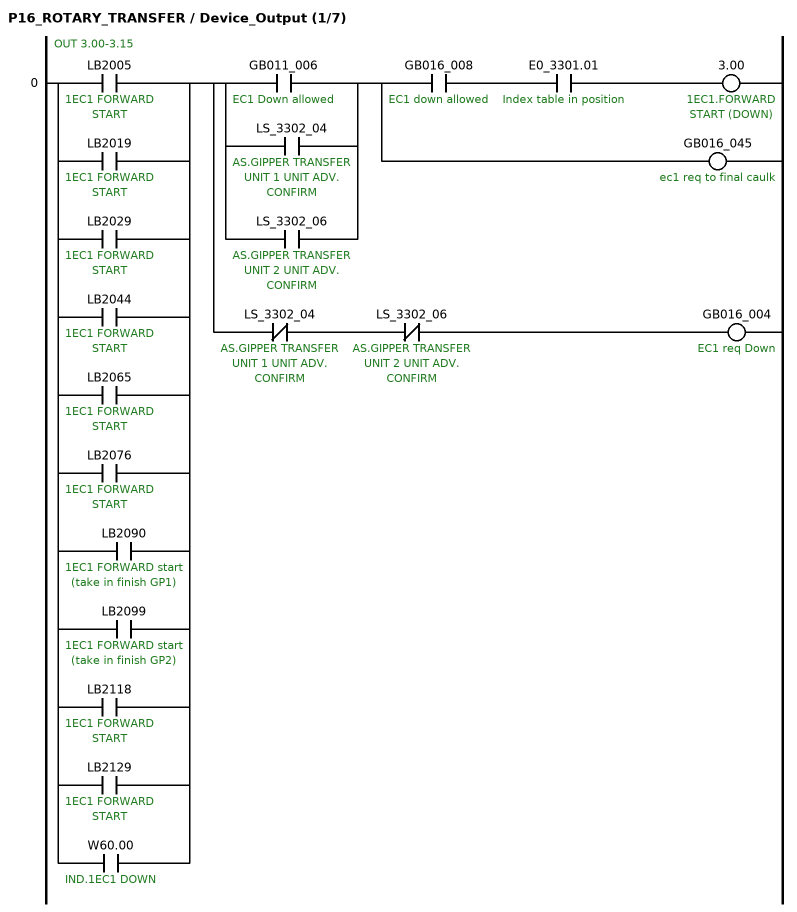
; [picture p264: P16_ROTARY_TRANSFER / Device_Output, rungs 0-0]
; rung 0: OUT 3.00-3.15
LD LB2005  ; 1EC1 FORWARD START
OR LB2019  ; 1EC1 FORWARD START
OR LB2029  ; 1EC1 FORWARD START
OR LB2044  ; 1EC1 FORWARD START
OR LB2065  ; 1EC1 FORWARD START
OR LB2076  ; 1EC1 FORWARD START
OR LB2090  ; 1EC1 FORWARD start (take in finish GP1)
OR LB2099  ; 1EC1 FORWARD start (take in finish GP2)
OR LB2118  ; 1EC1 FORWARD START
OR LB2129  ; 1EC1 FORWARD START
OR W60.00  ; IND.1EC1 DOWN
OUT TR0
LD GB011_006  ; EC1 Down allowed
OR LS_3302_04  ; AS.GIPPER TRANSFER UNIT 1 UNIT ADV. CONFIRM
OR LS_3302_06  ; AS.GIPPER TRANSFER UNIT 2 UNIT ADV. CONFIRM
ANDLD
OUT TR1
AND GB016_008  ; EC1 down allowed
AND E0_3301.01  ; Index table in position
OUT 3.00  ; 1EC1.FORWARD START (DOWN)
LD TR1
OUT GB016_045  ; ec1 req to final caulk
LD TR0
ANDNOT LS_3302_04  ; AS.GIPPER TRANSFER UNIT 1 UNIT ADV. CONFIRM
ANDNOT LS_3302_06  ; AS.GIPPER TRANSFER UNIT 2 UNIT ADV. CONFIRM
OUT GB016_004  ; EC1 req Down

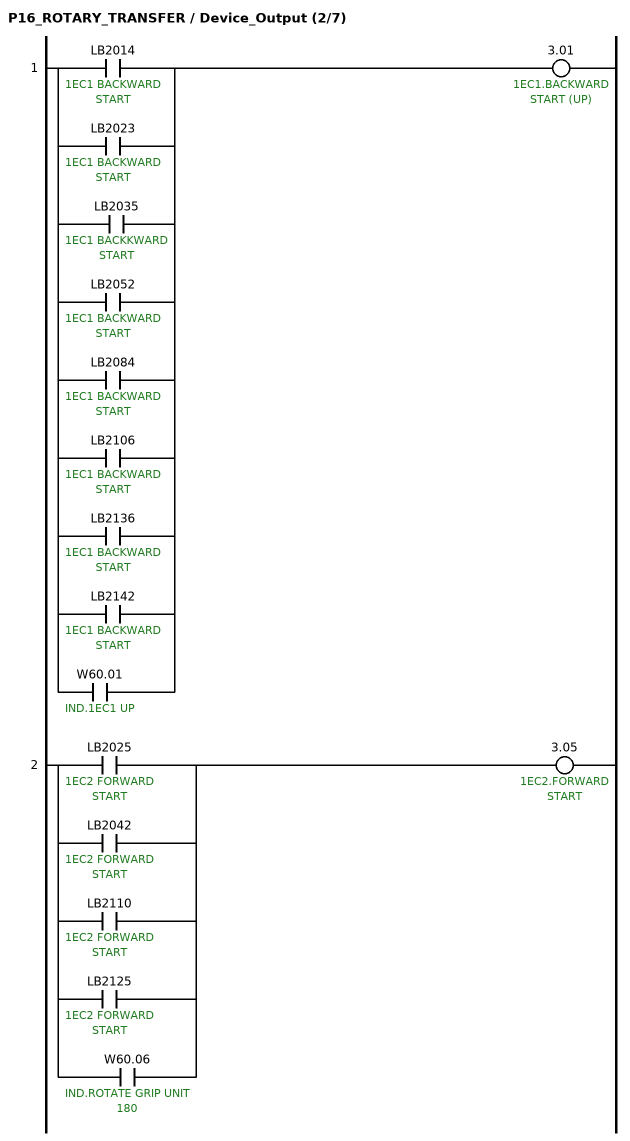
; rung 1
LD LB2014  ; 1EC1 BACKWARD START
OR LB2023  ; 1EC1 BACKWARD START
OR LB2035  ; 1EC1 BACKKWARD START
OR LB2052  ; 1EC1 BACKWARD START
OR LB2084  ; 1EC1 BACKWARD START
OR LB2106  ; 1EC1 BACKWARD START
OR LB2136  ; 1EC1 BACKWARD START
OR LB2142  ; 1EC1 BACKWARD START
OR W60.01  ; IND.1EC1 UP
OUT 3.01  ; 1EC1.BACKWARD START (UP)
; rung 2
LD LB2025  ; 1EC2 FORWARD START
OR LB2042  ; 1EC2 FORWARD START
OR LB2110  ; 1EC2 FORWARD START
OR LB2125  ; 1EC2 FORWARD START
OR W60.06  ; IND.ROTATE GRIP UNIT 180
OUT 3.05  ; 1EC2.FORWARD START

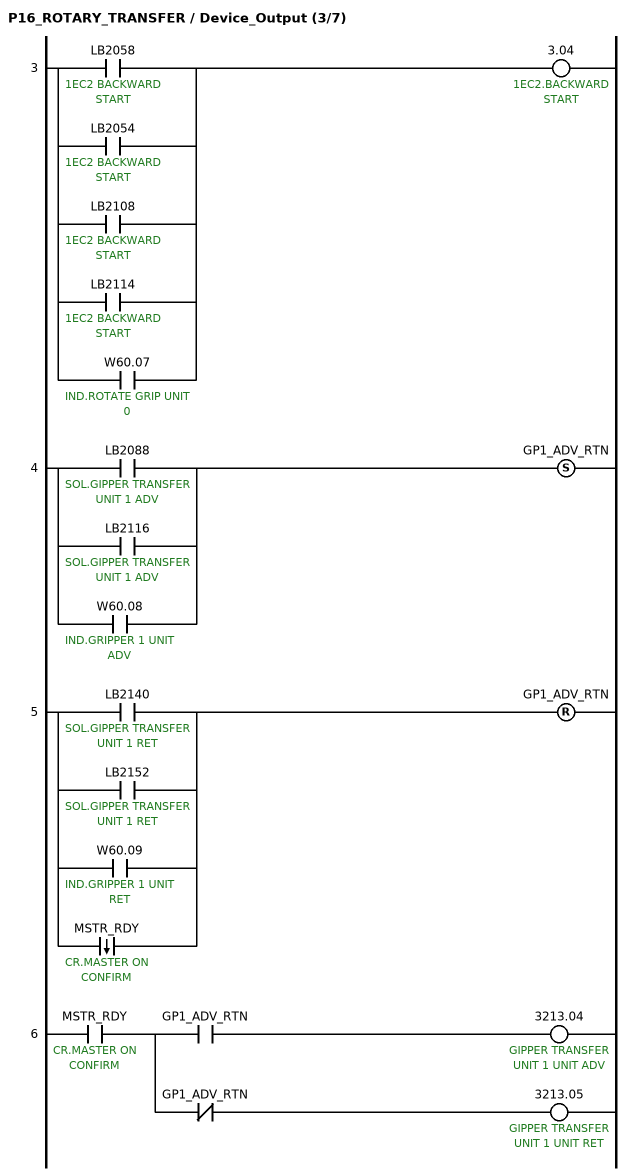
; rung 3
LD LB2058  ; 1EC2 BACKWARD START
OR LB2054  ; 1EC2 BACKWARD START
OR LB2108  ; 1EC2 BACKWARD START
OR LB2114  ; 1EC2 BACKWARD START
OR W60.07  ; IND.ROTATE GRIP UNIT 0
OUT 3.04  ; 1EC2.BACKWARD START
; rung 4
LD LB2088  ; SOL.GIPPER TRANSFER UNIT 1 ADV
OR LB2116  ; SOL.GIPPER TRANSFER UNIT 1 ADV
OR W60.08  ; IND.GRIPPER 1 UNIT ADV
SET GP1_ADV_RTN
; rung 5
LD LB2140  ; SOL.GIPPER TRANSFER UNIT 1 RET
OR LB2152  ; SOL.GIPPER TRANSFER UNIT 1 RET
OR W60.09  ; IND.GRIPPER 1 UNIT RET
%OR MSTR_RDY  ; CR.MASTER ON CONFIRM
RSET GP1_ADV_RTN
; rung 6
LD MSTR_RDY  ; CR.MASTER ON CONFIRM
OUT TR0
AND GP1_ADV_RTN
OUT 3213.04  ; GIPPER TRANSFER UNIT 1 UNIT ADV
LD TR0
ANDNOT GP1_ADV_RTN
OUT 3213.05  ; GIPPER TRANSFER UNIT 1 UNIT RET

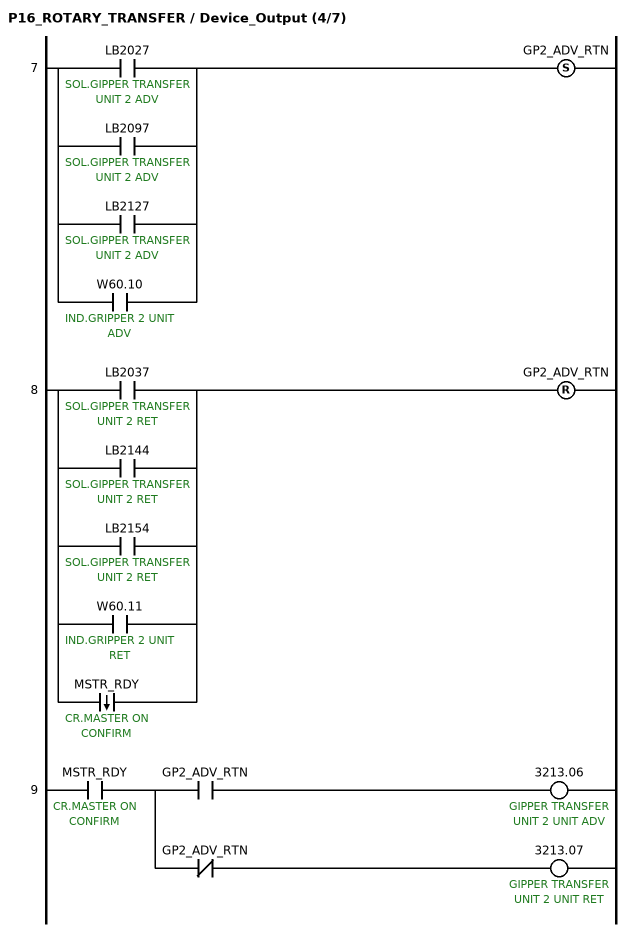
; rung 7
LD LB2027  ; SOL.GIPPER TRANSFER UNIT 2 ADV
OR LB2097  ; SOL.GIPPER TRANSFER UNIT 2 ADV
OR LB2127  ; SOL.GIPPER TRANSFER UNIT 2 ADV
OR W60.10  ; IND.GRIPPER 2 UNIT ADV
SET GP2_ADV_RTN
; rung 8
LD LB2037  ; SOL.GIPPER TRANSFER UNIT 2 RET
OR LB2144  ; SOL.GIPPER TRANSFER UNIT 2 RET
OR LB2154  ; SOL.GIPPER TRANSFER UNIT 2 RET
OR W60.11  ; IND.GRIPPER 2 UNIT RET
%OR MSTR_RDY  ; CR.MASTER ON CONFIRM
RSET GP2_ADV_RTN
; rung 9
LD MSTR_RDY  ; CR.MASTER ON CONFIRM
OUT TR0
AND GP2_ADV_RTN
OUT 3213.06  ; GIPPER TRANSFER UNIT 2 UNIT ADV
LD TR0
ANDNOT GP2_ADV_RTN
OUT 3213.07  ; GIPPER TRANSFER UNIT 2 UNIT RET

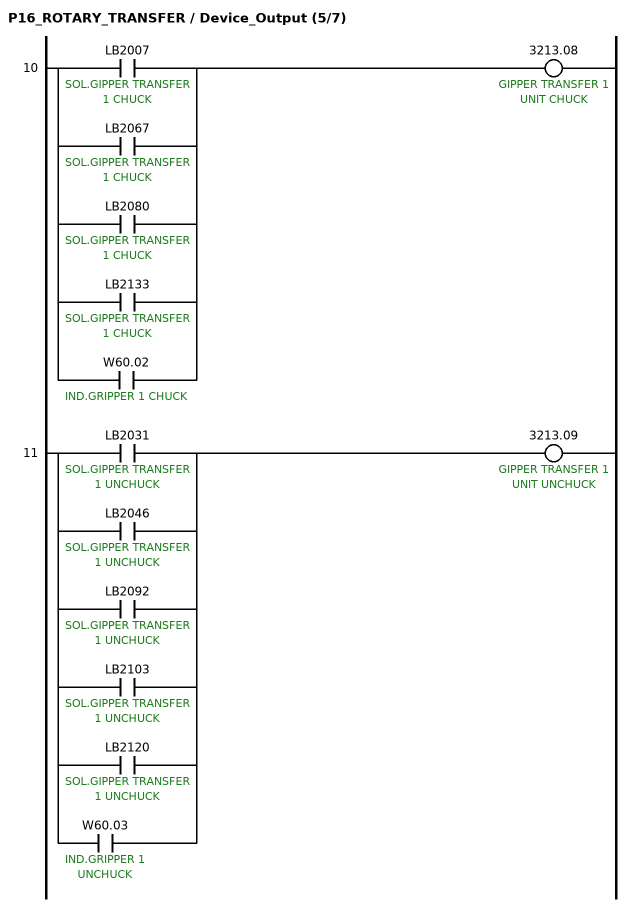
; rung 10
LD LB2007  ; SOL.GIPPER TRANSFER 1 CHUCK
OR LB2067  ; SOL.GIPPER TRANSFER 1 CHUCK
OR LB2080  ; SOL.GIPPER TRANSFER 1 CHUCK
OR LB2133  ; SOL.GIPPER TRANSFER 1 CHUCK
OR W60.02  ; IND.GRIPPER 1 CHUCK
OUT 3213.08  ; GIPPER TRANSFER 1 UNIT CHUCK
; rung 11
LD LB2031  ; SOL.GIPPER TRANSFER 1 UNCHUCK
OR LB2046  ; SOL.GIPPER TRANSFER 1 UNCHUCK
OR LB2092  ; SOL.GIPPER TRANSFER 1 UNCHUCK
OR LB2103  ; SOL.GIPPER TRANSFER 1 UNCHUCK
OR LB2120  ; SOL.GIPPER TRANSFER 1 UNCHUCK
OR W60.03  ; IND.GRIPPER 1 UNCHUCK
OUT 3213.09  ; GIPPER TRANSFER 1 UNIT UNCHUCK

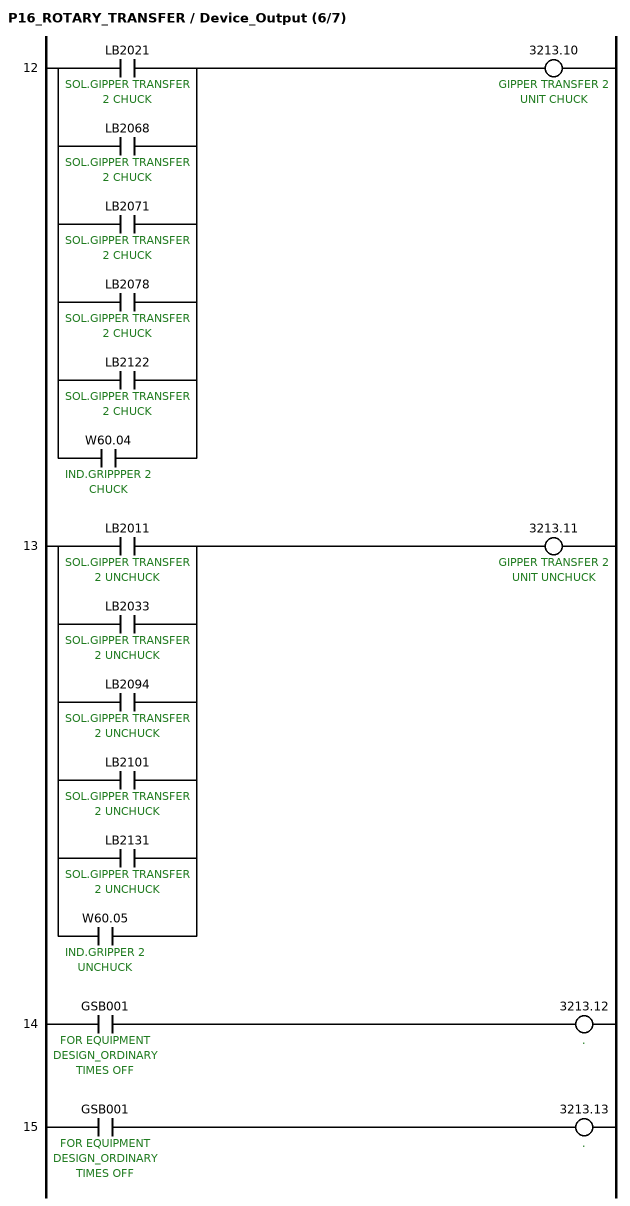
; rung 12
LD LB2021  ; SOL.GIPPER TRANSFER 2 CHUCK
OR LB2068  ; SOL.GIPPER TRANSFER 2 CHUCK
OR LB2071  ; SOL.GIPPER TRANSFER 2 CHUCK
OR LB2078  ; SOL.GIPPER TRANSFER 2 CHUCK
OR LB2122  ; SOL.GIPPER TRANSFER 2 CHUCK
OR W60.04  ; IND.GRIPPPER 2 CHUCK
OUT 3213.10  ; GIPPER TRANSFER 2 UNIT CHUCK
; rung 13
LD LB2011  ; SOL.GIPPER TRANSFER 2 UNCHUCK
OR LB2033  ; SOL.GIPPER TRANSFER 2 UNCHUCK
OR LB2094  ; SOL.GIPPER TRANSFER 2 UNCHUCK
OR LB2101  ; SOL.GIPPER TRANSFER 2 UNCHUCK
OR LB2131  ; SOL.GIPPER TRANSFER 2 UNCHUCK
OR W60.05  ; IND.GRIPPER 2 UNCHUCK
OUT 3213.11  ; GIPPER TRANSFER 2 UNIT UNCHUCK
; rung 14
LD GSB001  ; FOR EQUIPMENT DESIGN_ORDINARY TIMES OFF
OUT 3213.12  ; .
; rung 15
LD GSB001  ; FOR EQUIPMENT DESIGN_ORDINARY TIMES OFF
OUT 3213.13  ; .

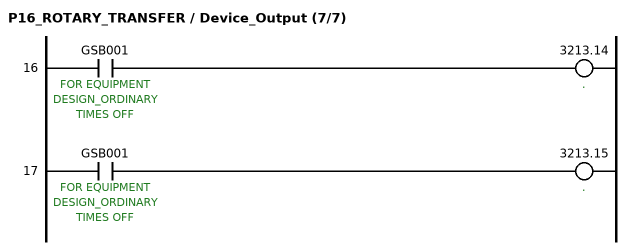
; rung 16
LD GSB001  ; FOR EQUIPMENT DESIGN_ORDINARY TIMES OFF
OUT 3213.14  ; .
; rung 17
LD GSB001  ; FOR EQUIPMENT DESIGN_ORDINARY TIMES OFF
OUT 3213.15  ; .

### Section Station_Output

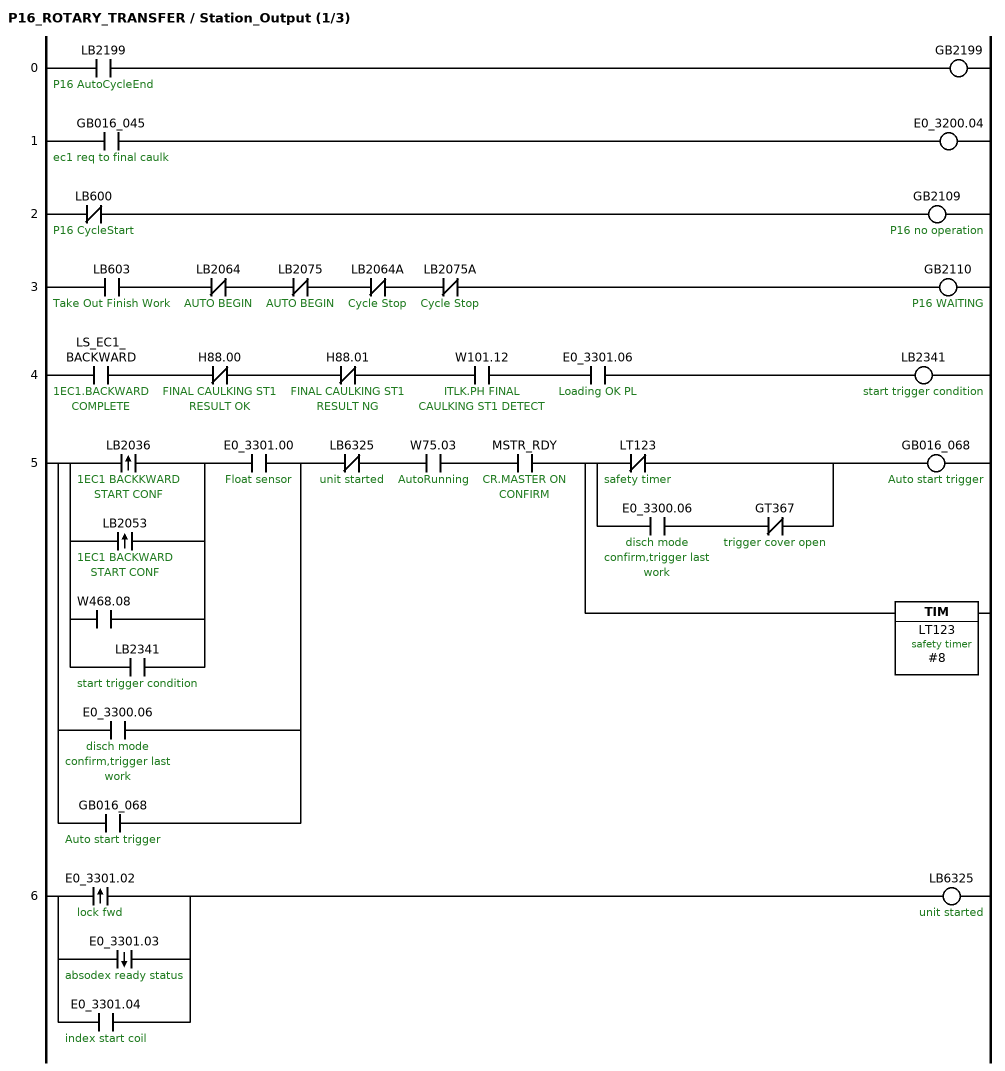
; rung 0
LD LB2199  ; P16 AutoCycleEnd
OUT GB2199
; rung 1
LD GB016_045  ; ec1 req to final caulk
OUT E0_3200.04
; rung 2
LDNOT LB600  ; P16 CycleStart
OUT GB2109  ; P16 no operation
; rung 3
LD LB603  ; Take Out Finish Work
ANDNOT LB2064  ; AUTO BEGIN
ANDNOT LB2075  ; AUTO BEGIN
ANDNOT LB2064A  ; Cycle Stop
ANDNOT LB2075A  ; Cycle Stop
OUT GB2110  ; P16 WAITING
; rung 4
LD LS_EC1_BACKWARD  ; 1EC1.BACKWARD COMPLETE
ANDNOT H88.00  ; FINAL CAULKING ST1 RESULT OK
ANDNOT H88.01  ; FINAL CAULKING ST1 RESULT NG
AND W101.12  ; ITLK.PH FINAL CAULKING ST1 DETECT
AND E0_3301.06  ; Loading OK PL
OUT LB2341  ; start trigger condition
; rung 5
@LD LB2036  ; 1EC1 BACKKWARD START CONF
@OR LB2053  ; 1EC1 BACKWARD START CONF
OR W468.08
OR LB2341  ; start trigger condition
AND E0_3301.00  ; Float sensor
OR E0_3300.06  ; disch mode confirm,trigger last work
OR GB016_068  ; Auto start trigger
ANDNOT LB6325  ; unit started
AND W75.03  ; AutoRunning
AND MSTR_RDY  ; CR.MASTER ON CONFIRM
OUT TR0
LDNOT LT123  ; safety timer
LD E0_3300.06  ; disch mode confirm,trigger last work
ANDNOT GT367  ; trigger cover open
ORLD
ANDLD
OUT GB016_068  ; Auto start trigger
LD TR0
TIM LT123 #8  ; safety timer
; rung 6
@LD E0_3301.02  ; lock fwd
%OR E0_3301.03  ; absodex ready status
OR E0_3301.04  ; index start coil
OUT LB6325  ; unit started

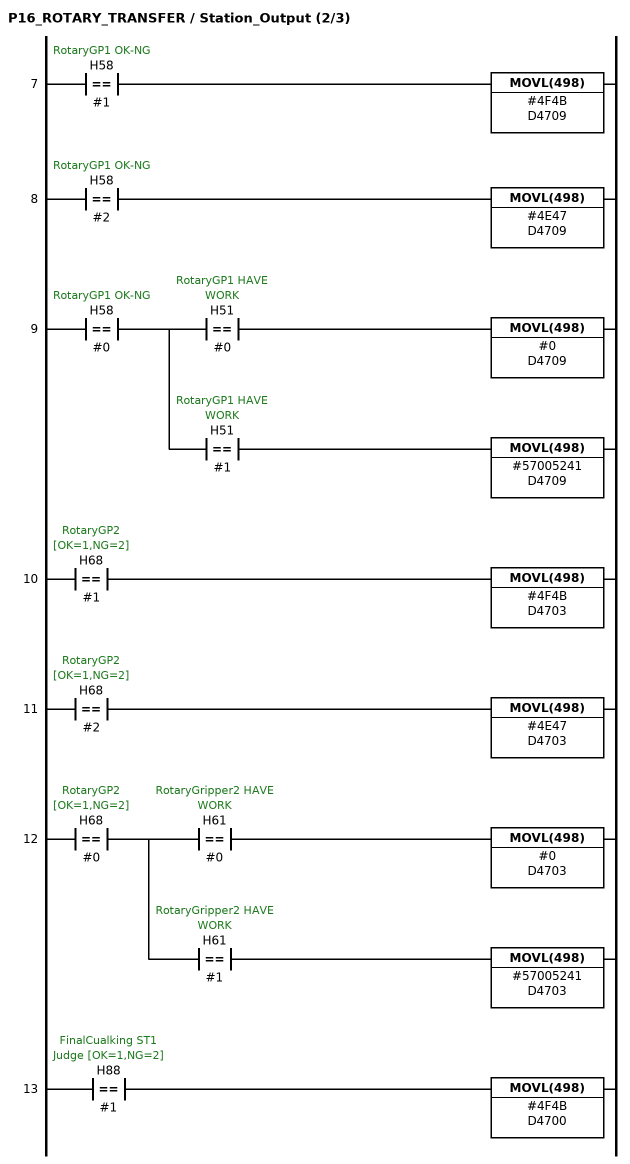
; rung 7
LD=(300) H58 #1  ; RotaryGP1 OK-NG
MOVL(498) #4F4B D4709
; rung 8
LD=(300) H58 #2  ; RotaryGP1 OK-NG
MOVL(498) #4E47 D4709
; rung 9
LD=(300) H58 #0  ; RotaryGP1 OK-NG
OUT TR0
AND=(300) H51 #0  ; RotaryGP1 HAVE WORK
MOVL(498) #0 D4709
LD TR0
AND=(300) H51 #1  ; RotaryGP1 HAVE WORK
MOVL(498) #57005241 D4709
; rung 10
LD=(300) H68 #1  ; RotaryGP2 [OK=1,NG=2]
MOVL(498) #4F4B D4703
; rung 11
LD=(300) H68 #2  ; RotaryGP2 [OK=1,NG=2]
MOVL(498) #4E47 D4703
; rung 12
LD=(300) H68 #0  ; RotaryGP2 [OK=1,NG=2]
OUT TR0
AND=(300) H61 #0  ; RotaryGripper2 HAVE WORK
MOVL(498) #0 D4703
LD TR0
AND=(300) H61 #1  ; RotaryGripper2 HAVE WORK
MOVL(498) #57005241 D4703
; rung 13
LD=(300) H88 #1  ; FinalCualking ST1 Judge [OK=1,NG=2]
MOVL(498) #4F4B D4700

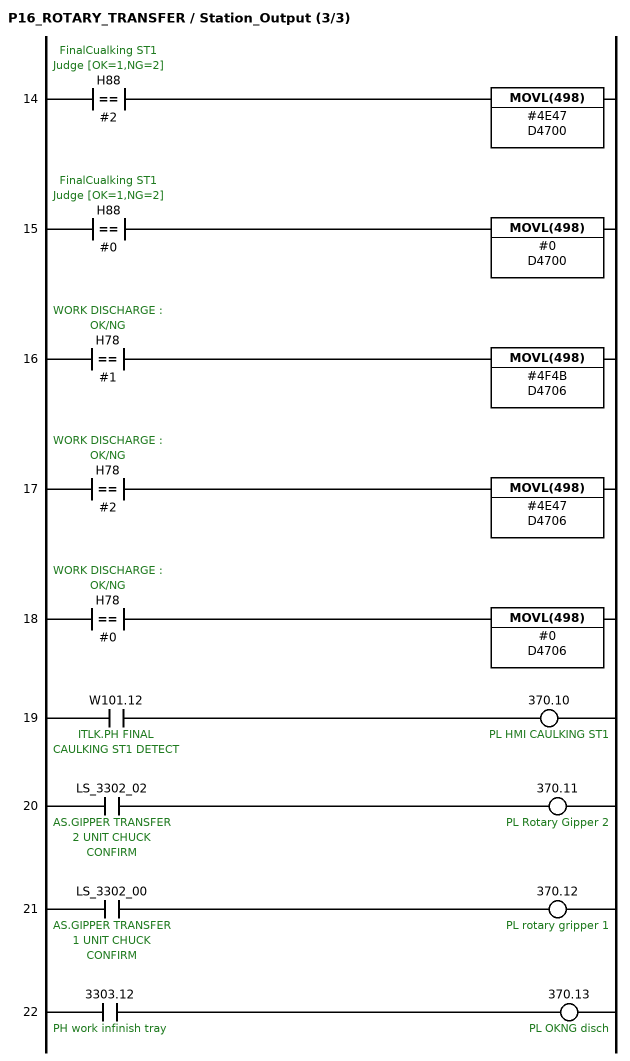
; rung 14
LD=(300) H88 #2  ; FinalCualking ST1 Judge [OK=1,NG=2]
MOVL(498) #4E47 D4700
; rung 15
LD=(300) H88 #0  ; FinalCualking ST1 Judge [OK=1,NG=2]
MOVL(498) #0 D4700
; rung 16
LD=(300) H78 #1  ; WORK DISCHARGE : OK/NG
MOVL(498) #4F4B D4706
; rung 17
LD=(300) H78 #2  ; WORK DISCHARGE : OK/NG
MOVL(498) #4E47 D4706
; rung 18
LD=(300) H78 #0  ; WORK DISCHARGE : OK/NG
MOVL(498) #0 D4706
; rung 19
LD W101.12  ; ITLK.PH FINAL CAULKING ST1 DETECT
OUT 370.10  ; PL HMI CAULKING ST1
; rung 20
LD LS_3302_02  ; AS.GIPPER TRANSFER 2 UNIT CHUCK CONFIRM
OUT 370.11  ; PL Rotary Gipper 2
; rung 21
LD LS_3302_00  ; AS.GIPPER TRANSFER 1 UNIT CHUCK CONFIRM
OUT 370.12  ; PL rotary gripper 1
; rung 22
LD 3303.12  ; PH work infinish tray
OUT 370.13  ; PL OKNG disch

### Section Individual

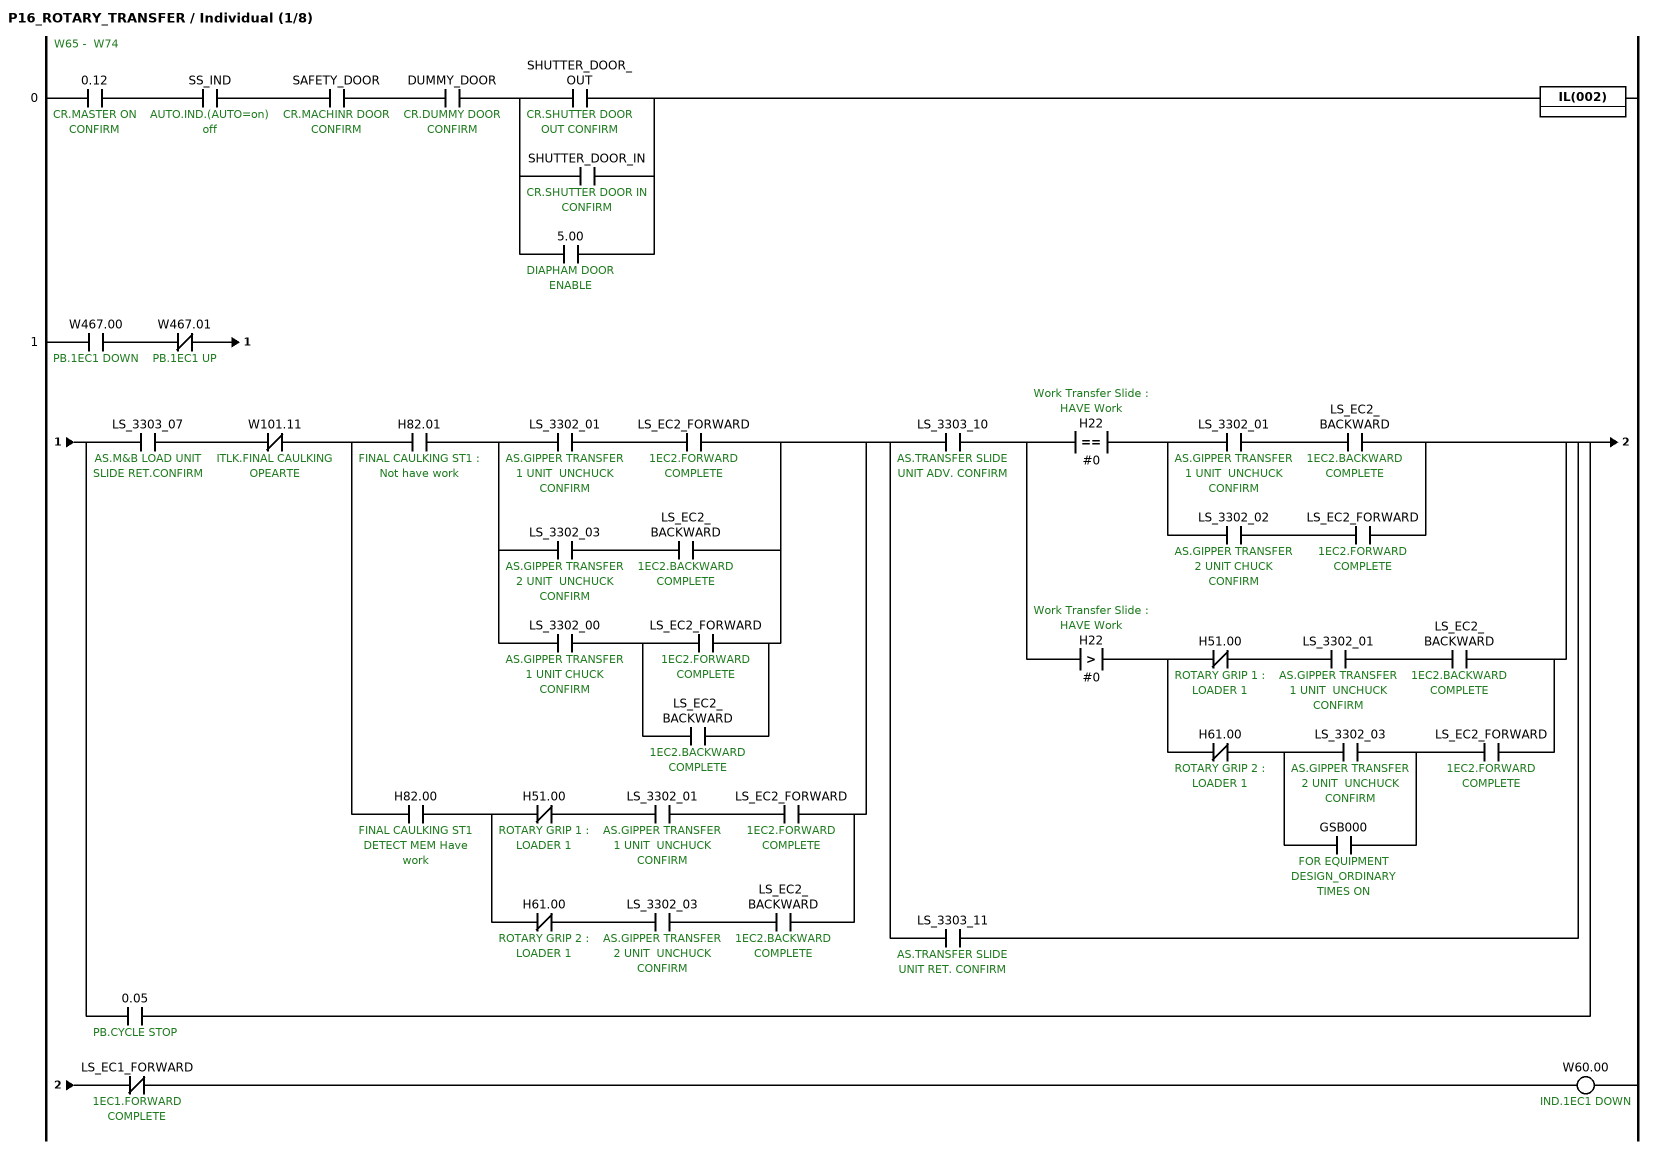
; rung 0: W65 -  W74
LD 0.12  ; CR.MASTER ON CONFIRM
AND SS_IND  ; AUTO.IND.(AUTO=on) off
AND SAFETY_DOOR  ; CR.MACHINR DOOR CONFIRM
AND DUMMY_DOOR  ; CR.DUMMY DOOR CONFIRM
LD SHUTTER_DOOR_OUT  ; CR.SHUTTER DOOR OUT CONFIRM
OR SHUTTER_DOOR_IN  ; CR.SHUTTER DOOR IN CONFIRM
OR 5.00  ; DIAPHAM DOOR ENABLE
ANDLD
IL(002)
; rung 1
LD W467.00  ; PB.1EC1 DOWN
ANDNOT W467.01  ; PB.1EC1 UP
LD LS_3303_07  ; AS.M&B LOAD UNIT SLIDE RET.CONFIRM
ANDNOT W101.11  ; ITLK.FINAL CAULKING OPEARTE
LD H82.01  ; FINAL CAULKING ST1 : Not have work
LD LS_3302_01  ; AS.GIPPER TRANSFER 1 UNIT  UNCHUCK CONFIRM
AND LS_EC2_FORWARD  ; 1EC2.FORWARD COMPLETE
LD LS_3302_03  ; AS.GIPPER TRANSFER 2 UNIT  UNCHUCK CONFIRM
AND LS_EC2_BACKWARD  ; 1EC2.BACKWARD COMPLETE
ORLD
LD LS_3302_00  ; AS.GIPPER TRANSFER 1 UNIT CHUCK CONFIRM
LD LS_EC2_FORWARD  ; 1EC2.FORWARD COMPLETE
OR LS_EC2_BACKWARD  ; 1EC2.BACKWARD COMPLETE
ANDLD
ORLD
ANDLD
LD H82.00  ; FINAL CAULKING ST1 DETECT MEM Have work
LDNOT H51.00  ; ROTARY GRIP 1 : LOADER 1
AND LS_3302_01  ; AS.GIPPER TRANSFER 1 UNIT  UNCHUCK CONFIRM
AND LS_EC2_FORWARD  ; 1EC2.FORWARD COMPLETE
LDNOT H61.00  ; ROTARY GRIP 2 : LOADER 1
AND LS_3302_03  ; AS.GIPPER TRANSFER 2 UNIT  UNCHUCK CONFIRM
AND LS_EC2_BACKWARD  ; 1EC2.BACKWARD COMPLETE
ORLD
ANDLD
ORLD
ANDLD
LD LS_3303_10  ; AS.TRANSFER SLIDE UNIT ADV. CONFIRM
LD=(300) H22 #0  ; Work Transfer Slide : HAVE Work
LD LS_3302_01  ; AS.GIPPER TRANSFER 1 UNIT  UNCHUCK CONFIRM
AND LS_EC2_BACKWARD  ; 1EC2.BACKWARD COMPLETE
LD LS_3302_02  ; AS.GIPPER TRANSFER 2 UNIT CHUCK CONFIRM
AND LS_EC2_FORWARD  ; 1EC2.FORWARD COMPLETE
ORLD
ANDLD
LD>(320) H22 #0  ; Work Transfer Slide : HAVE Work
LDNOT H51.00  ; ROTARY GRIP 1 : LOADER 1
AND LS_3302_01  ; AS.GIPPER TRANSFER 1 UNIT  UNCHUCK CONFIRM
AND LS_EC2_BACKWARD  ; 1EC2.BACKWARD COMPLETE
LDNOT H61.00  ; ROTARY GRIP 2 : LOADER 1
LD LS_3302_03  ; AS.GIPPER TRANSFER 2 UNIT  UNCHUCK CONFIRM
OR GSB000  ; FOR EQUIPMENT DESIGN_ORDINARY TIMES ON
ANDLD
AND LS_EC2_FORWARD  ; 1EC2.FORWARD COMPLETE
ORLD
ANDLD
ORLD
ANDLD
OR LS_3303_11  ; AS.TRANSFER SLIDE UNIT RET. CONFIRM
ANDLD
OR 0.05  ; PB.CYCLE STOP
ANDLD
ANDNOT LS_EC1_FORWARD  ; 1EC1.FORWARD COMPLETE
OUT W60.00  ; IND.1EC1 DOWN

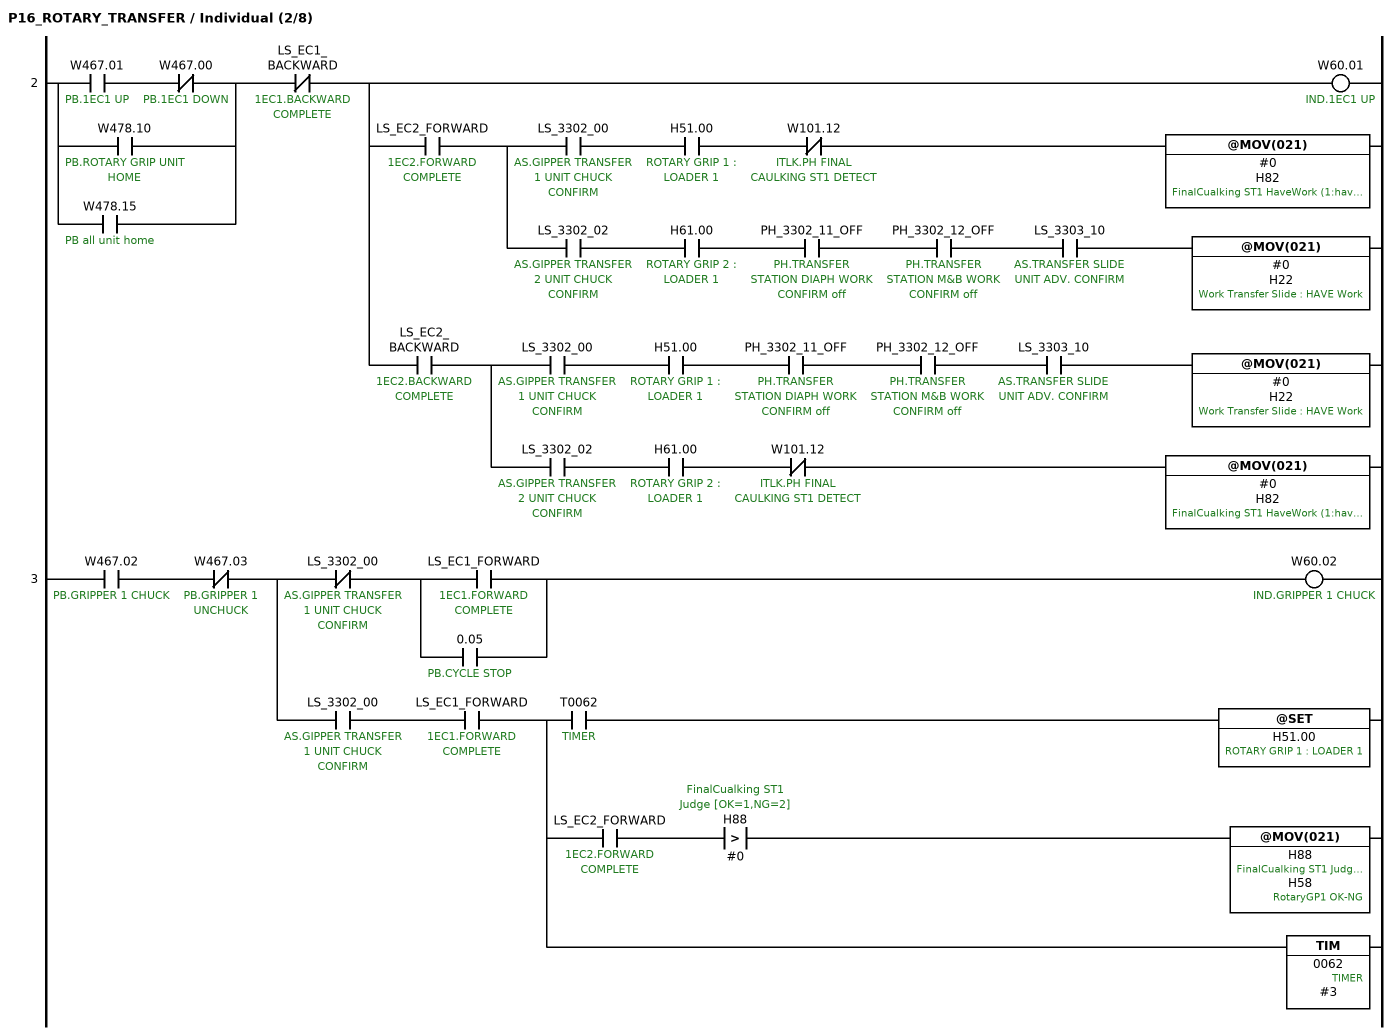
; rung 2
LD W467.01  ; PB.1EC1 UP
ANDNOT W467.00  ; PB.1EC1 DOWN
LD W478.10  ; PB.ROTARY GRIP UNIT HOME
OR W478.15  ; PB all unit home
ORLD
ANDNOT LS_EC1_BACKWARD  ; 1EC1.BACKWARD COMPLETE
OUT TR0
OUT W60.01  ; IND.1EC1 UP
AND LS_EC2_FORWARD  ; 1EC2.FORWARD COMPLETE
OUT TR1
AND LS_3302_00  ; AS.GIPPER TRANSFER 1 UNIT CHUCK CONFIRM
AND H51.00  ; ROTARY GRIP 1 : LOADER 1
ANDNOT W101.12  ; ITLK.PH FINAL CAULKING ST1 DETECT
@MOV(021) #0 H82  ; FinalCualking ST1 HaveWork (1:have work 2:no work)
LD TR1
AND LS_3302_02  ; AS.GIPPER TRANSFER 2 UNIT CHUCK CONFIRM
AND H61.00  ; ROTARY GRIP 2 : LOADER 1
AND PH_3302_11_OFF  ; PH.TRANSFER STATION DIAPH WORK CONFIRM off
AND PH_3302_12_OFF  ; PH.TRANSFER STATION M&B WORK CONFIRM off
AND LS_3303_10  ; AS.TRANSFER SLIDE UNIT ADV. CONFIRM
@MOV(021) #0 H22  ; Work Transfer Slide : HAVE Work
LD TR0
AND LS_EC2_BACKWARD  ; 1EC2.BACKWARD COMPLETE
OUT TR0
AND LS_3302_00  ; AS.GIPPER TRANSFER 1 UNIT CHUCK CONFIRM
AND H51.00  ; ROTARY GRIP 1 : LOADER 1
AND PH_3302_11_OFF  ; PH.TRANSFER STATION DIAPH WORK CONFIRM off
AND PH_3302_12_OFF  ; PH.TRANSFER STATION M&B WORK CONFIRM off
AND LS_3303_10  ; AS.TRANSFER SLIDE UNIT ADV. CONFIRM
@MOV(021) #0 H22  ; Work Transfer Slide : HAVE Work
LD TR0
AND LS_3302_02  ; AS.GIPPER TRANSFER 2 UNIT CHUCK CONFIRM
AND H61.00  ; ROTARY GRIP 2 : LOADER 1
ANDNOT W101.12  ; ITLK.PH FINAL CAULKING ST1 DETECT
@MOV(021) #0 H82  ; FinalCualking ST1 HaveWork (1:have work 2:no work)
; rung 3
LD W467.02  ; PB.GRIPPER 1 CHUCK
ANDNOT W467.03  ; PB.GRIPPER 1 UNCHUCK
OUT TR0
ANDNOT LS_3302_00  ; AS.GIPPER TRANSFER 1 UNIT CHUCK CONFIRM
LD LS_EC1_FORWARD  ; 1EC1.FORWARD COMPLETE
OR 0.05  ; PB.CYCLE STOP
ANDLD
OUT W60.02  ; IND.GRIPPER 1 CHUCK
LD TR0
AND LS_3302_00  ; AS.GIPPER TRANSFER 1 UNIT CHUCK CONFIRM
AND LS_EC1_FORWARD  ; 1EC1.FORWARD COMPLETE
OUT TR0
AND T0062  ; TIMER
@SET H51.00  ; ROTARY GRIP 1 : LOADER 1
LD TR0
AND LS_EC2_FORWARD  ; 1EC2.FORWARD COMPLETE
AND>(320) H88 #0  ; FinalCualking ST1 Judge [OK=1,NG=2]
@MOV(021) H88 H58  ; FinalCualking ST1 Judge [OK=1,NG=2], RotaryGP1 OK-NG
LD TR0
TIM 0062 #3  ; TIMER

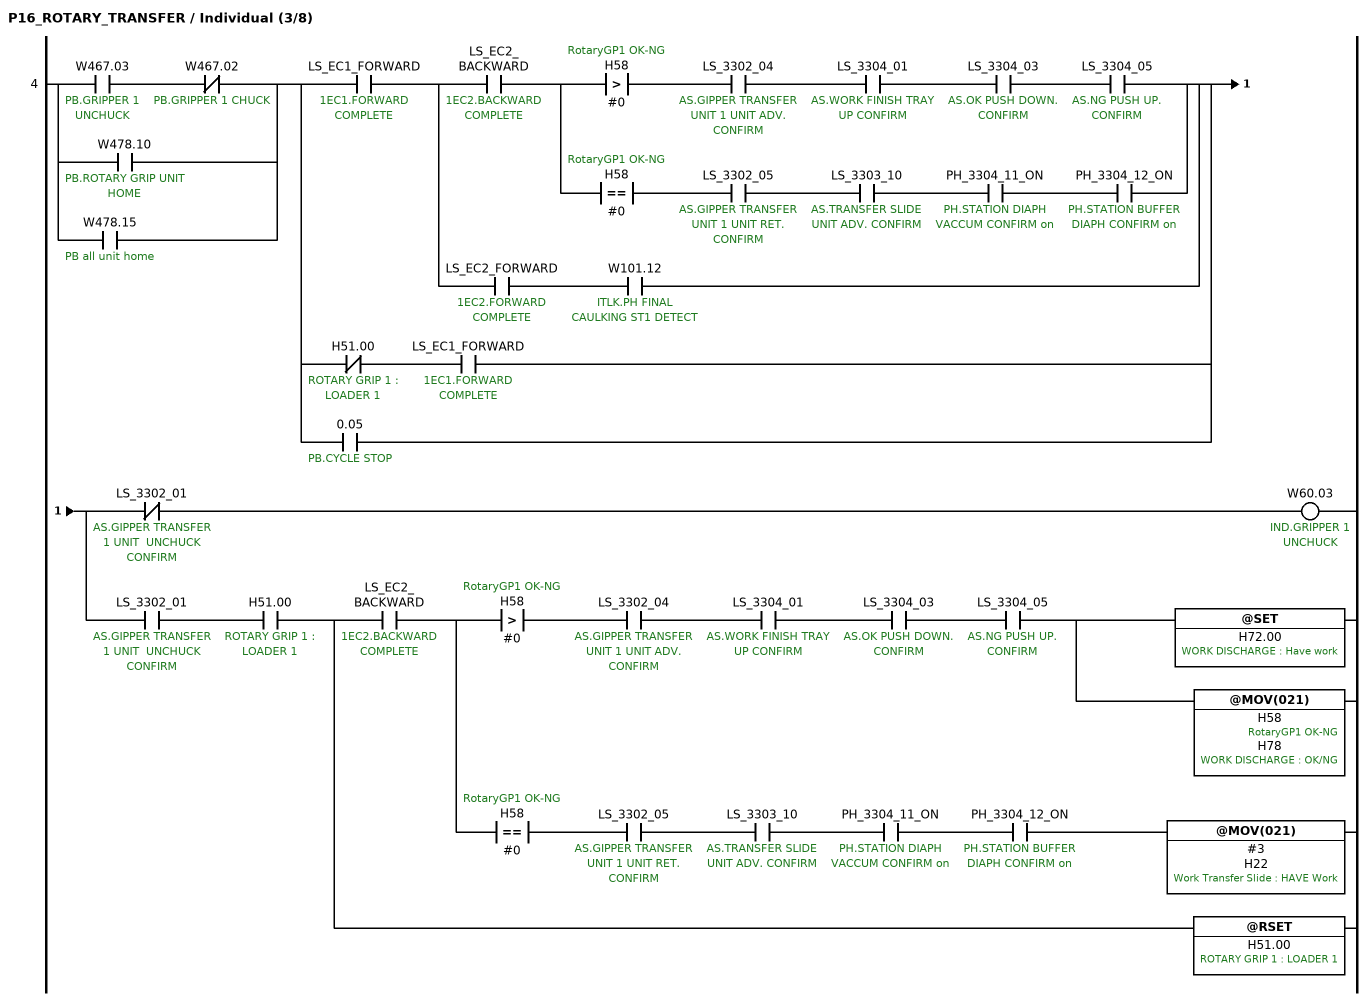
; rung 4
LD W467.03  ; PB.GRIPPER 1 UNCHUCK
ANDNOT W467.02  ; PB.GRIPPER 1 CHUCK
OR W478.10  ; PB.ROTARY GRIP UNIT HOME
OR W478.15  ; PB all unit home
LD LS_EC1_FORWARD  ; 1EC1.FORWARD COMPLETE
LD LS_EC2_BACKWARD  ; 1EC2.BACKWARD COMPLETE
LD>(320) H58 #0  ; RotaryGP1 OK-NG
AND LS_3302_04  ; AS.GIPPER TRANSFER UNIT 1 UNIT ADV. CONFIRM
AND LS_3304_01  ; AS.WORK FINISH TRAY UP CONFIRM
AND LS_3304_03  ; AS.OK PUSH DOWN. CONFIRM
AND LS_3304_05  ; AS.NG PUSH UP. CONFIRM
LD=(300) H58 #0  ; RotaryGP1 OK-NG
AND LS_3302_05  ; AS.GIPPER TRANSFER UNIT 1 UNIT RET. CONFIRM
AND LS_3303_10  ; AS.TRANSFER SLIDE UNIT ADV. CONFIRM
AND PH_3304_11_ON  ; PH.STATION DIAPH VACCUM CONFIRM on
AND PH_3304_12_ON  ; PH.STATION BUFFER DIAPH CONFIRM on
ORLD
ANDLD
LD LS_EC2_FORWARD  ; 1EC2.FORWARD COMPLETE
AND W101.12  ; ITLK.PH FINAL CAULKING ST1 DETECT
ORLD
ANDLD
LDNOT H51.00  ; ROTARY GRIP 1 : LOADER 1
AND LS_EC1_FORWARD  ; 1EC1.FORWARD COMPLETE
ORLD
OR 0.05  ; PB.CYCLE STOP
ANDLD
OUT TR0
ANDNOT LS_3302_01  ; AS.GIPPER TRANSFER 1 UNIT  UNCHUCK CONFIRM
OUT W60.03  ; IND.GRIPPER 1 UNCHUCK
LD TR0
AND LS_3302_01  ; AS.GIPPER TRANSFER 1 UNIT  UNCHUCK CONFIRM
AND H51.00  ; ROTARY GRIP 1 : LOADER 1
OUT TR0
AND LS_EC2_BACKWARD  ; 1EC2.BACKWARD COMPLETE
OUT TR1
AND>(320) H58 #0  ; RotaryGP1 OK-NG
AND LS_3302_04  ; AS.GIPPER TRANSFER UNIT 1 UNIT ADV. CONFIRM
AND LS_3304_01  ; AS.WORK FINISH TRAY UP CONFIRM
AND LS_3304_03  ; AS.OK PUSH DOWN. CONFIRM
AND LS_3304_05  ; AS.NG PUSH UP. CONFIRM
@SET H72.00  ; WORK DISCHARGE : Have work
@MOV(021) H58 H78  ; RotaryGP1 OK-NG, WORK DISCHARGE : OK/NG
LD TR1
AND=(300) H58 #0  ; RotaryGP1 OK-NG
AND LS_3302_05  ; AS.GIPPER TRANSFER UNIT 1 UNIT RET. CONFIRM
AND LS_3303_10  ; AS.TRANSFER SLIDE UNIT ADV. CONFIRM
AND PH_3304_11_ON  ; PH.STATION DIAPH VACCUM CONFIRM on
AND PH_3304_12_ON  ; PH.STATION BUFFER DIAPH CONFIRM on
@MOV(021) #3 H22  ; Work Transfer Slide : HAVE Work
LD TR0
@RSET H51.00  ; ROTARY GRIP 1 : LOADER 1

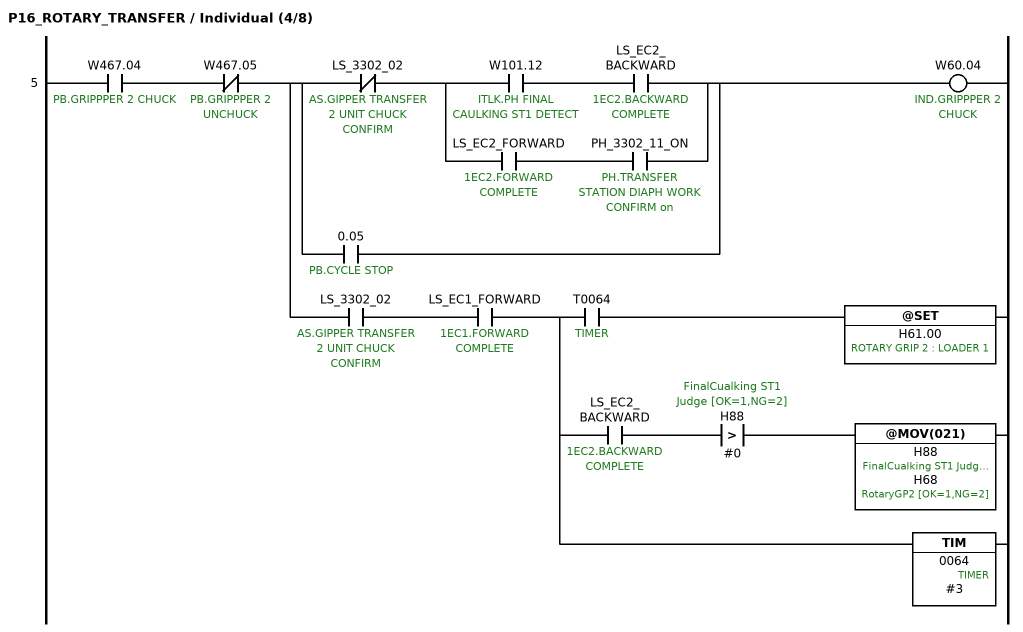
; rung 5
LD W467.04  ; PB.GRIPPPER 2 CHUCK
ANDNOT W467.05  ; PB.GRIPPPER 2 UNCHUCK
OUT TR0
LDNOT LS_3302_02  ; AS.GIPPER TRANSFER 2 UNIT CHUCK CONFIRM
LD W101.12  ; ITLK.PH FINAL CAULKING ST1 DETECT
AND LS_EC2_BACKWARD  ; 1EC2.BACKWARD COMPLETE
LD LS_EC2_FORWARD  ; 1EC2.FORWARD COMPLETE
AND PH_3302_11_ON  ; PH.TRANSFER STATION DIAPH WORK CONFIRM on
ORLD
ANDLD
OR 0.05  ; PB.CYCLE STOP
ANDLD
OUT W60.04  ; IND.GRIPPPER 2 CHUCK
LD TR0
AND LS_3302_02  ; AS.GIPPER TRANSFER 2 UNIT CHUCK CONFIRM
AND LS_EC1_FORWARD  ; 1EC1.FORWARD COMPLETE
OUT TR0
AND T0064  ; TIMER
@SET H61.00  ; ROTARY GRIP 2 : LOADER 1
LD TR0
AND LS_EC2_BACKWARD  ; 1EC2.BACKWARD COMPLETE
AND>(320) H88 #0  ; FinalCualking ST1 Judge [OK=1,NG=2]
@MOV(021) H88 H68  ; FinalCualking ST1 Judge [OK=1,NG=2], RotaryGP2 [OK=1,NG=2]
LD TR0
TIM 0064 #3  ; TIMER

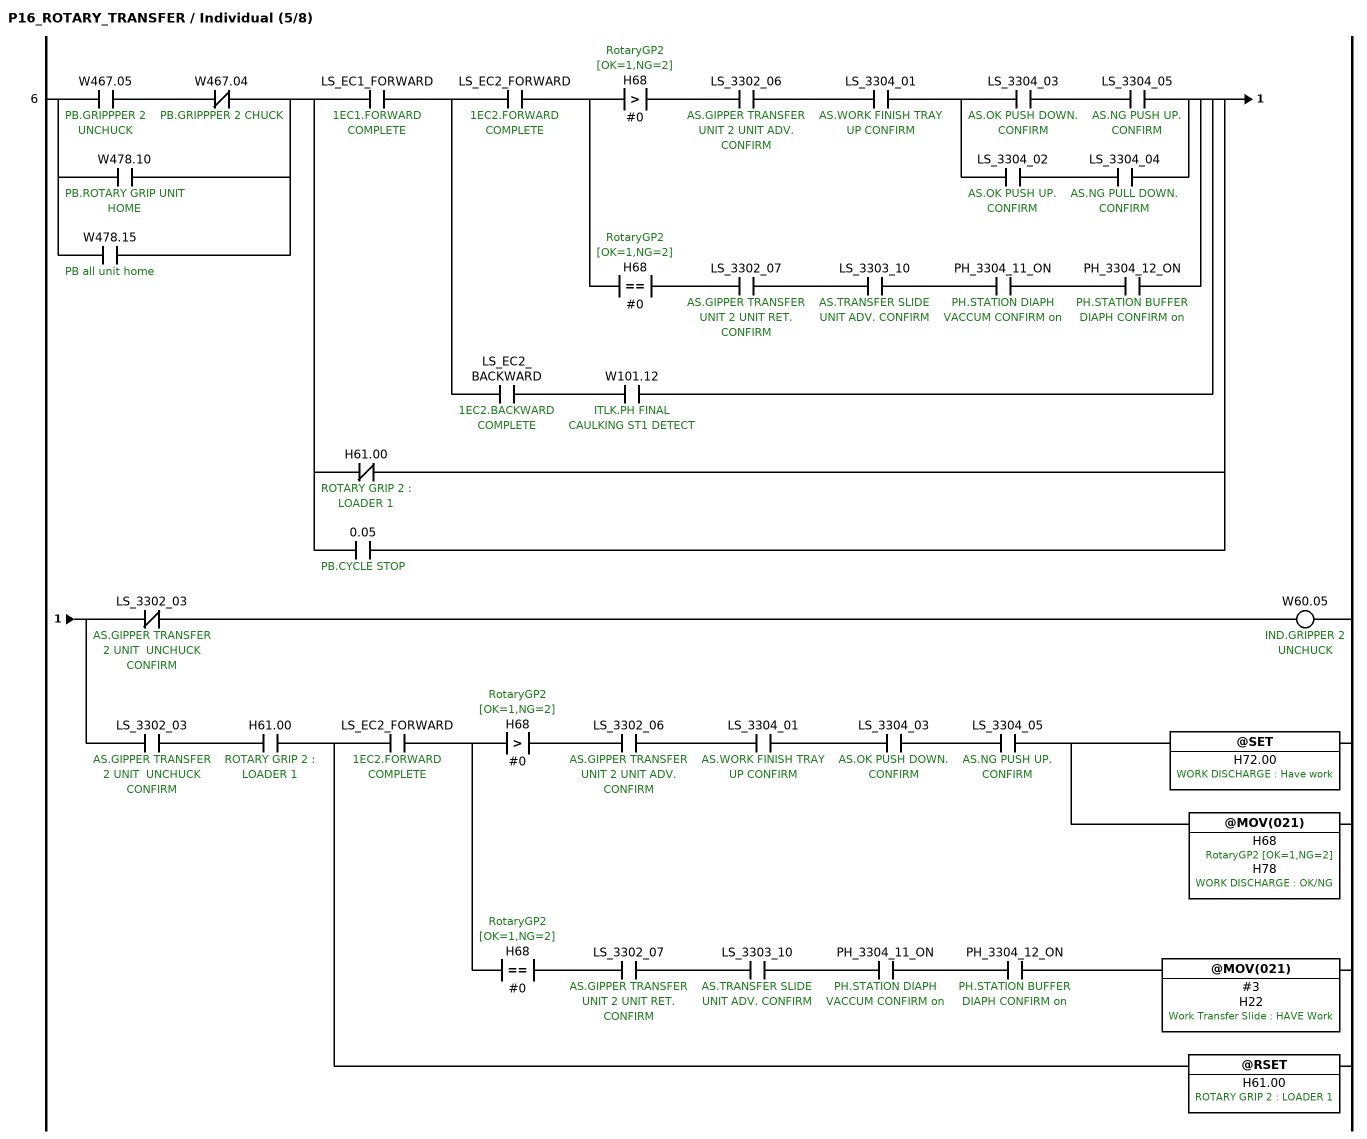
; rung 6
LD W467.05  ; PB.GRIPPPER 2 UNCHUCK
ANDNOT W467.04  ; PB.GRIPPPER 2 CHUCK
LD W478.10  ; PB.ROTARY GRIP UNIT HOME
OR W478.15  ; PB all unit home
ORLD
LD LS_EC1_FORWARD  ; 1EC1.FORWARD COMPLETE
LD LS_EC2_FORWARD  ; 1EC2.FORWARD COMPLETE
LD>(320) H68 #0  ; RotaryGP2 [OK=1,NG=2]
AND LS_3302_06  ; AS.GIPPER TRANSFER UNIT 2 UNIT ADV. CONFIRM
AND LS_3304_01  ; AS.WORK FINISH TRAY UP CONFIRM
LD LS_3304_03  ; AS.OK PUSH DOWN. CONFIRM
AND LS_3304_05  ; AS.NG PUSH UP. CONFIRM
LD LS_3304_02  ; AS.OK PUSH UP. CONFIRM
AND LS_3304_04  ; AS.NG PULL DOWN. CONFIRM
ORLD
ANDLD
LD=(300) H68 #0  ; RotaryGP2 [OK=1,NG=2]
AND LS_3302_07  ; AS.GIPPER TRANSFER UNIT 2 UNIT RET. CONFIRM
AND LS_3303_10  ; AS.TRANSFER SLIDE UNIT ADV. CONFIRM
AND PH_3304_11_ON  ; PH.STATION DIAPH VACCUM CONFIRM on
AND PH_3304_12_ON  ; PH.STATION BUFFER DIAPH CONFIRM on
ORLD
ANDLD
LD LS_EC2_BACKWARD  ; 1EC2.BACKWARD COMPLETE
AND W101.12  ; ITLK.PH FINAL CAULKING ST1 DETECT
ORLD
ANDLD
ORNOT H61.00  ; ROTARY GRIP 2 : LOADER 1
OR 0.05  ; PB.CYCLE STOP
ANDLD
OUT TR0
ANDNOT LS_3302_03  ; AS.GIPPER TRANSFER 2 UNIT  UNCHUCK CONFIRM
OUT W60.05  ; IND.GRIPPER 2 UNCHUCK
LD TR0
AND LS_3302_03  ; AS.GIPPER TRANSFER 2 UNIT  UNCHUCK CONFIRM
AND H61.00  ; ROTARY GRIP 2 : LOADER 1
OUT TR0
AND LS_EC2_FORWARD  ; 1EC2.FORWARD COMPLETE
OUT TR1
AND>(320) H68 #0  ; RotaryGP2 [OK=1,NG=2]
AND LS_3302_06  ; AS.GIPPER TRANSFER UNIT 2 UNIT ADV. CONFIRM
AND LS_3304_01  ; AS.WORK FINISH TRAY UP CONFIRM
AND LS_3304_03  ; AS.OK PUSH DOWN. CONFIRM
AND LS_3304_05  ; AS.NG PUSH UP. CONFIRM
@SET H72.00  ; WORK DISCHARGE : Have work
@MOV(021) H68 H78  ; RotaryGP2 [OK=1,NG=2], WORK DISCHARGE : OK/NG
LD TR1
AND=(300) H68 #0  ; RotaryGP2 [OK=1,NG=2]
AND LS_3302_07  ; AS.GIPPER TRANSFER UNIT 2 UNIT RET. CONFIRM
AND LS_3303_10  ; AS.TRANSFER SLIDE UNIT ADV. CONFIRM
AND PH_3304_11_ON  ; PH.STATION DIAPH VACCUM CONFIRM on
AND PH_3304_12_ON  ; PH.STATION BUFFER DIAPH CONFIRM on
@MOV(021) #3 H22  ; Work Transfer Slide : HAVE Work
LD TR0
@RSET H61.00  ; ROTARY GRIP 2 : LOADER 1

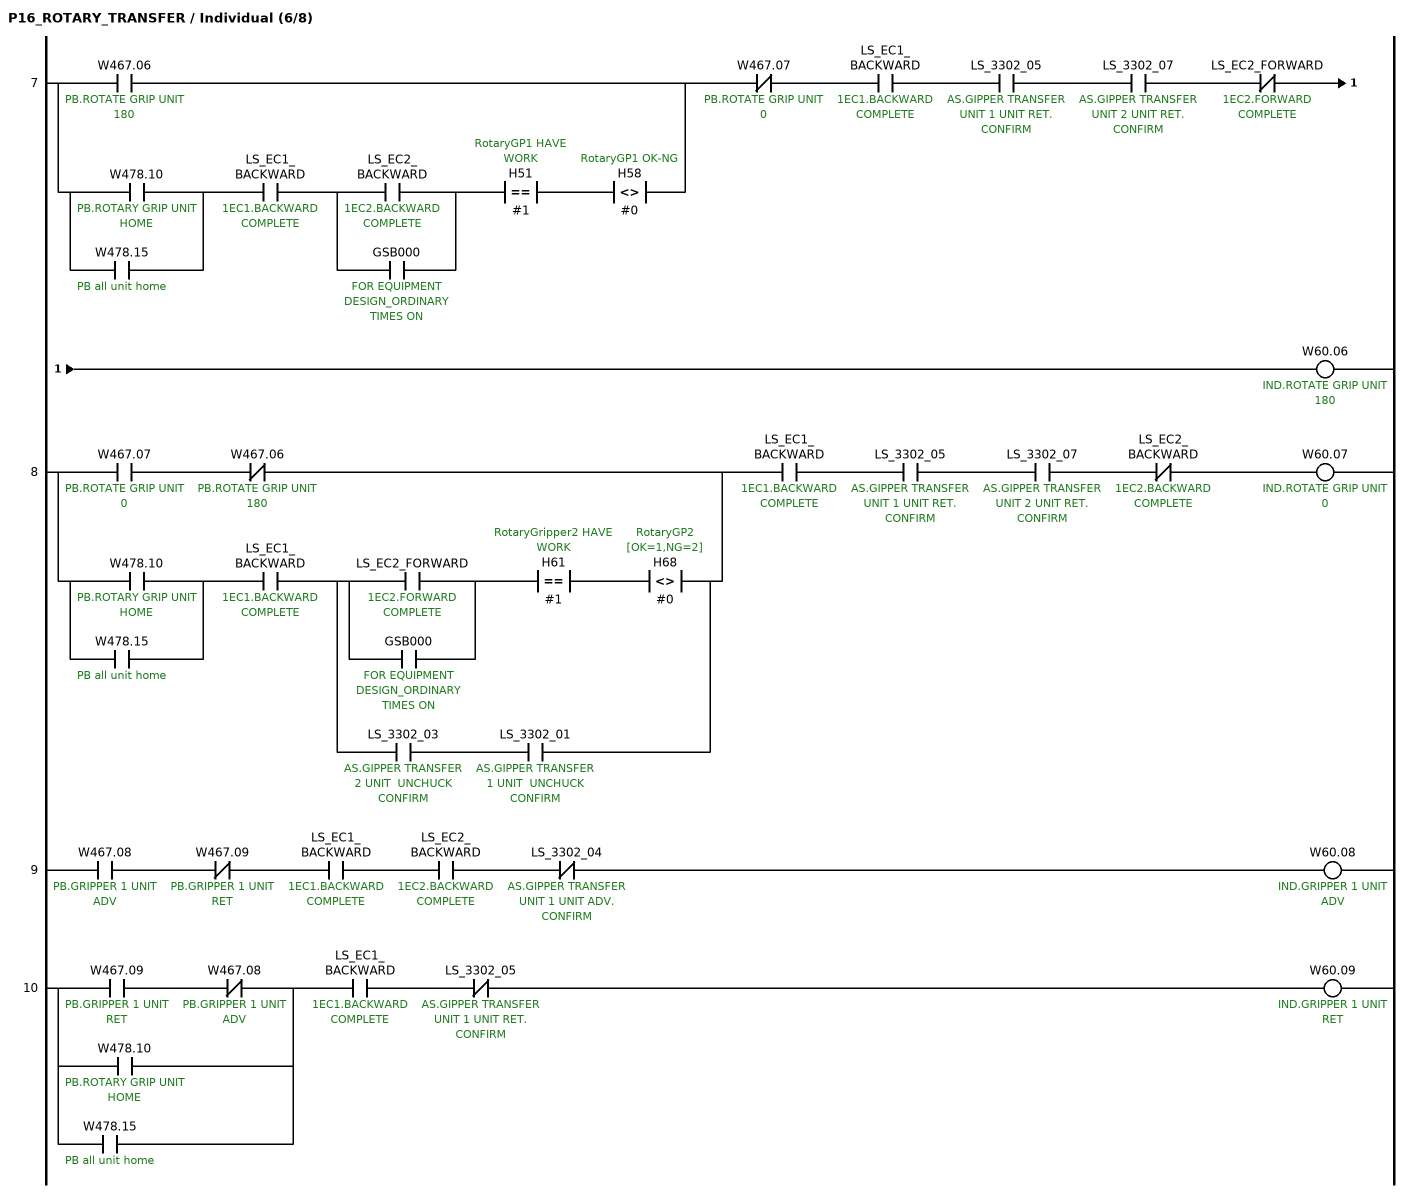
; rung 7
LD W467.06  ; PB.ROTATE GRIP UNIT 180
LD W478.10  ; PB.ROTARY GRIP UNIT HOME
OR W478.15  ; PB all unit home
AND LS_EC1_BACKWARD  ; 1EC1.BACKWARD COMPLETE
LD LS_EC2_BACKWARD  ; 1EC2.BACKWARD COMPLETE
OR GSB000  ; FOR EQUIPMENT DESIGN_ORDINARY TIMES ON
ANDLD
AND=(300) H51 #1  ; RotaryGP1 HAVE WORK
AND<>(305) H58 #0  ; RotaryGP1 OK-NG
ORLD
ANDNOT W467.07  ; PB.ROTATE GRIP UNIT 0
AND LS_EC1_BACKWARD  ; 1EC1.BACKWARD COMPLETE
AND LS_3302_05  ; AS.GIPPER TRANSFER UNIT 1 UNIT RET. CONFIRM
AND LS_3302_07  ; AS.GIPPER TRANSFER UNIT 2 UNIT RET. CONFIRM
ANDNOT LS_EC2_FORWARD  ; 1EC2.FORWARD COMPLETE
OUT W60.06  ; IND.ROTATE GRIP UNIT 180
; rung 8
LD W467.07  ; PB.ROTATE GRIP UNIT 0
ANDNOT W467.06  ; PB.ROTATE GRIP UNIT 180
LD W478.10  ; PB.ROTARY GRIP UNIT HOME
OR W478.15  ; PB all unit home
AND LS_EC1_BACKWARD  ; 1EC1.BACKWARD COMPLETE
LD LS_EC2_FORWARD  ; 1EC2.FORWARD COMPLETE
OR GSB000  ; FOR EQUIPMENT DESIGN_ORDINARY TIMES ON
AND=(300) H61 #1  ; RotaryGripper2 HAVE WORK
AND<>(305) H68 #0  ; RotaryGP2 [OK=1,NG=2]
LD LS_3302_03  ; AS.GIPPER TRANSFER 2 UNIT  UNCHUCK CONFIRM
AND LS_3302_01  ; AS.GIPPER TRANSFER 1 UNIT  UNCHUCK CONFIRM
ORLD
ANDLD
ORLD
AND LS_EC1_BACKWARD  ; 1EC1.BACKWARD COMPLETE
AND LS_3302_05  ; AS.GIPPER TRANSFER UNIT 1 UNIT RET. CONFIRM
AND LS_3302_07  ; AS.GIPPER TRANSFER UNIT 2 UNIT RET. CONFIRM
ANDNOT LS_EC2_BACKWARD  ; 1EC2.BACKWARD COMPLETE
OUT W60.07  ; IND.ROTATE GRIP UNIT 0
; rung 9
LD W467.08  ; PB.GRIPPER 1 UNIT ADV
ANDNOT W467.09  ; PB.GRIPPER 1 UNIT RET
AND LS_EC1_BACKWARD  ; 1EC1.BACKWARD COMPLETE
AND LS_EC2_BACKWARD  ; 1EC2.BACKWARD COMPLETE
ANDNOT LS_3302_04  ; AS.GIPPER TRANSFER UNIT 1 UNIT ADV. CONFIRM
OUT W60.08  ; IND.GRIPPER 1 UNIT ADV
; rung 10
LD W467.09  ; PB.GRIPPER 1 UNIT RET
ANDNOT W467.08  ; PB.GRIPPER 1 UNIT ADV
LD W478.10  ; PB.ROTARY GRIP UNIT HOME
OR W478.15  ; PB all unit home
ORLD
AND LS_EC1_BACKWARD  ; 1EC1.BACKWARD COMPLETE
ANDNOT LS_3302_05  ; AS.GIPPER TRANSFER UNIT 1 UNIT RET. CONFIRM
OUT W60.09  ; IND.GRIPPER 1 UNIT RET

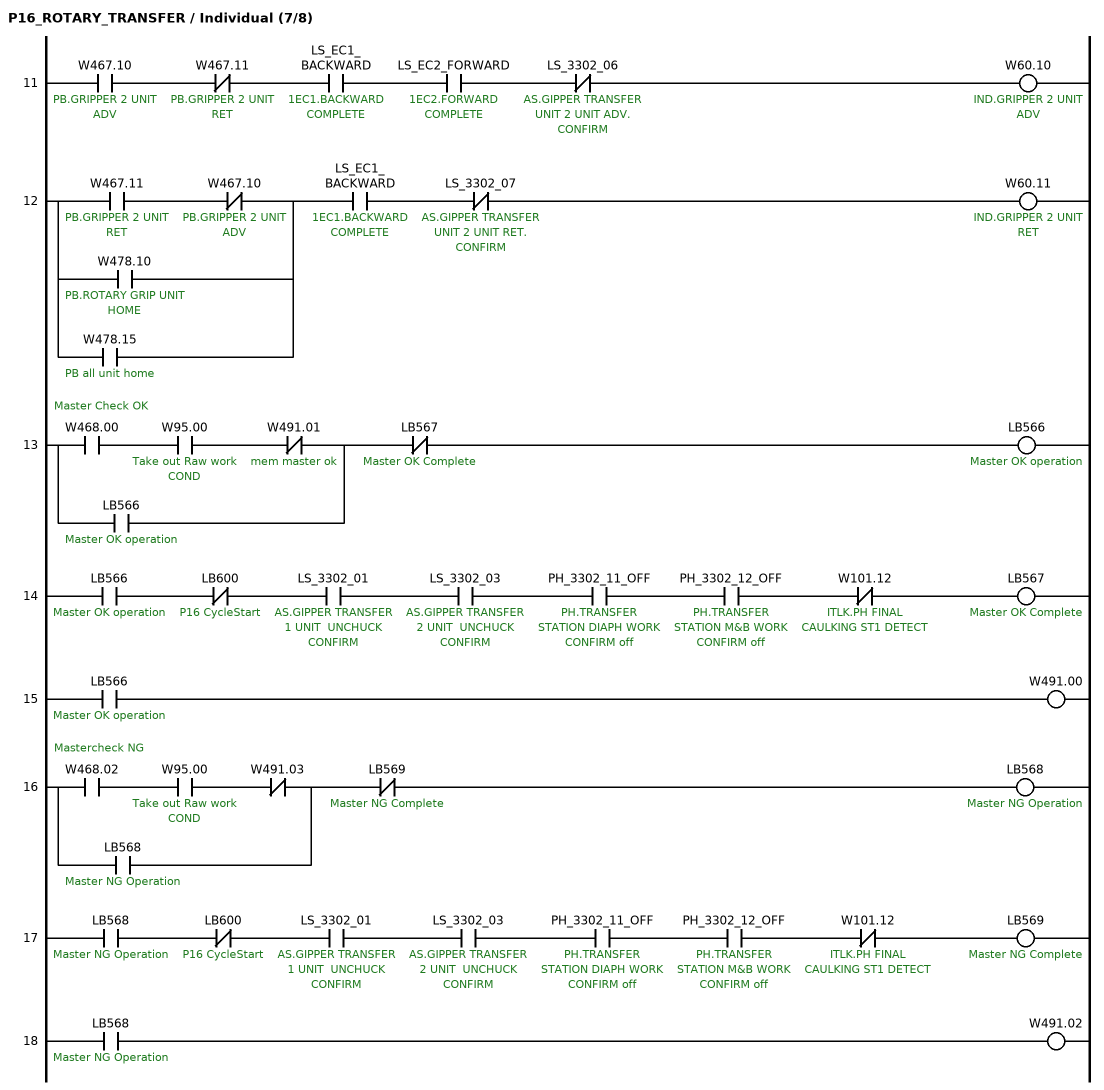
; rung 11
LD W467.10  ; PB.GRIPPER 2 UNIT ADV
ANDNOT W467.11  ; PB.GRIPPER 2 UNIT RET
AND LS_EC1_BACKWARD  ; 1EC1.BACKWARD COMPLETE
AND LS_EC2_FORWARD  ; 1EC2.FORWARD COMPLETE
ANDNOT LS_3302_06  ; AS.GIPPER TRANSFER UNIT 2 UNIT ADV. CONFIRM
OUT W60.10  ; IND.GRIPPER 2 UNIT ADV
; rung 12
LD W467.11  ; PB.GRIPPER 2 UNIT RET
ANDNOT W467.10  ; PB.GRIPPER 2 UNIT ADV
LD W478.10  ; PB.ROTARY GRIP UNIT HOME
OR W478.15  ; PB all unit home
ORLD
AND LS_EC1_BACKWARD  ; 1EC1.BACKWARD COMPLETE
ANDNOT LS_3302_07  ; AS.GIPPER TRANSFER UNIT 2 UNIT RET. CONFIRM
OUT W60.11  ; IND.GRIPPER 2 UNIT RET
; rung 13: Master Check OK
LD W468.00
AND W95.00  ; Take out Raw work COND
ANDNOT W491.01  ; mem master ok
OR LB566  ; Master OK operation
ANDNOT LB567  ; Master OK Complete
OUT LB566  ; Master OK operation
; rung 14
LD LB566  ; Master OK operation
ANDNOT LB600  ; P16 CycleStart
AND LS_3302_01  ; AS.GIPPER TRANSFER 1 UNIT  UNCHUCK CONFIRM
AND LS_3302_03  ; AS.GIPPER TRANSFER 2 UNIT  UNCHUCK CONFIRM
AND PH_3302_11_OFF  ; PH.TRANSFER STATION DIAPH WORK CONFIRM off
AND PH_3302_12_OFF  ; PH.TRANSFER STATION M&B WORK CONFIRM off
ANDNOT W101.12  ; ITLK.PH FINAL CAULKING ST1 DETECT
OUT LB567  ; Master OK Complete
; rung 15
LD LB566  ; Master OK operation
OUT W491.00
; rung 16: Mastercheck NG
LD W468.02
AND W95.00  ; Take out Raw work COND
ANDNOT W491.03
OR LB568  ; Master NG Operation
ANDNOT LB569  ; Master NG Complete
OUT LB568  ; Master NG Operation
; rung 17
LD LB568  ; Master NG Operation
ANDNOT LB600  ; P16 CycleStart
AND LS_3302_01  ; AS.GIPPER TRANSFER 1 UNIT  UNCHUCK CONFIRM
AND LS_3302_03  ; AS.GIPPER TRANSFER 2 UNIT  UNCHUCK CONFIRM
AND PH_3302_11_OFF  ; PH.TRANSFER STATION DIAPH WORK CONFIRM off
AND PH_3302_12_OFF  ; PH.TRANSFER STATION M&B WORK CONFIRM off
ANDNOT W101.12  ; ITLK.PH FINAL CAULKING ST1 DETECT
OUT LB569  ; Master NG Complete
; rung 18
LD LB568  ; Master NG Operation
OUT W491.02

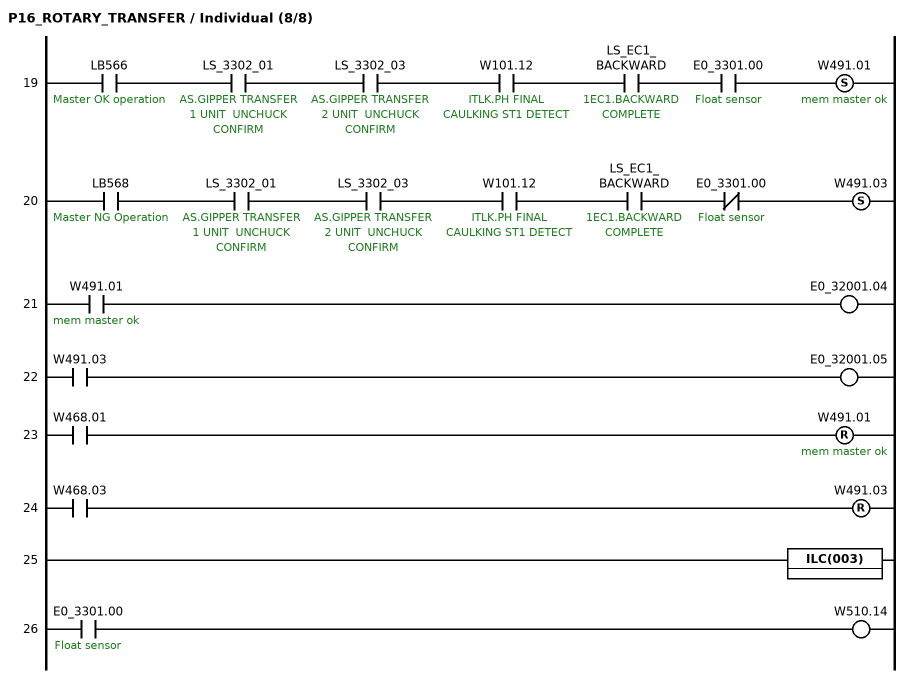
; rung 19
LD LB566  ; Master OK operation
AND LS_3302_01  ; AS.GIPPER TRANSFER 1 UNIT  UNCHUCK CONFIRM
AND LS_3302_03  ; AS.GIPPER TRANSFER 2 UNIT  UNCHUCK CONFIRM
AND W101.12  ; ITLK.PH FINAL CAULKING ST1 DETECT
AND LS_EC1_BACKWARD  ; 1EC1.BACKWARD COMPLETE
AND E0_3301.00  ; Float sensor
SET W491.01  ; mem master ok
; rung 20
LD LB568  ; Master NG Operation
AND LS_3302_01  ; AS.GIPPER TRANSFER 1 UNIT  UNCHUCK CONFIRM
AND LS_3302_03  ; AS.GIPPER TRANSFER 2 UNIT  UNCHUCK CONFIRM
AND W101.12  ; ITLK.PH FINAL CAULKING ST1 DETECT
AND LS_EC1_BACKWARD  ; 1EC1.BACKWARD COMPLETE
ANDNOT E0_3301.00  ; Float sensor
SET W491.03
; rung 21
LD W491.01  ; mem master ok
OUT E0_32001.04
; rung 22
LD W491.03
OUT E0_32001.05
; rung 23
LD W468.01
RSET W491.01  ; mem master ok
; rung 24
LD W468.03
RSET W491.03
; rung 25
ILC(003)
; rung 26
LD E0_3301.00  ; Float sensor
OUT W510.14

### Section END
; rung 0
END(001)

## Program P17_OK_NG_DISCHARGE (cyclic task 7)
Local symbols
LB2199 E0_46.15 BOOL  ; P16 AutoCycleEnd
LB2200 E0_41.02 BOOL  ; AUTO START BEGIN
LB2201 E0_41.03 BOOL  ; SOL.WORK FINISH TRAY DOWN
LB2202 E0_41.04 BOOL  ; SOL.WORK FINISH TRAY DOWN CONF
LB2203 E0_41.05 BOOL  ; SOL.OK PUSH UP
LB2204 E0_41.06 BOOL  ; SOL.OK PUSH UP CONF
LB2205 E0_41.07 BOOL  ; OK DISCHARGE CONFIRM
LB2206 E0_41.08 BOOL  ; SOL.OK PUSH DOWN
LB2207 E0_41.09 BOOL  ; SOL.OK PUSH DOWN CONF
LB2208 E0_41.10 BOOL  ; SOL.WORK FINISH TRAY UP
LB2209 E0_41.11 BOOL  ; SOL.WORK FINISH TRAY UP CONF
LB2210 E0_41.12 BOOL  ; AUTO START BEGIN
LB2211 E0_41.13 BOOL  ; SOL.WORK FINISH TRAY DOWN
LB2212 E0_41.14 BOOL  ; SOL.WORK FINISH TRAY DOWN CONF
LB2213 E0_41.15 BOOL  ; SOL.NG PUSH DOWN
LB2214 E0_42.00 BOOL  ; SOL.NG PUSH DOWN CONF
LB2215 E0_42.01 BOOL  ; NG DISCHARGE CONFIRM
LB2216 E0_42.02 BOOL  ; SOL.NG PUSH UP
LB2217 E0_42.03 BOOL  ; SOL.NG PUSH UP CONF
LB2218 E0_42.04 BOOL  ; SOL.WORK FINISH TRAY UP
LB2219 E0_42.05 BOOL  ; SOL.WORK FINISH TRAY UP CONF
LB2397 E0_42.06 BOOL  ; P16 OK Discharge END
LB2398 E0_42.07 BOOL  ; P16 NG Discharge END
LB2399 E0_42.08 BOOL  ; P17 AutoCycleEnd
LB432 E0_47.00 BOOL  ; IND 1 CYCLE
LB700 E0_42.09 BOOL  ; P17 CycleStart
LB701 E0_42.10 BOOL  ; P17 OK Discharge
LB702 E0_42.11 BOOL  ; P17 NG Discharge
LT2214 T3020 TIMER
LT231 T3024 TIMER
LT232 T3028 TIMER
trial_cv E0_46.02 BOOL

### Section Autorun

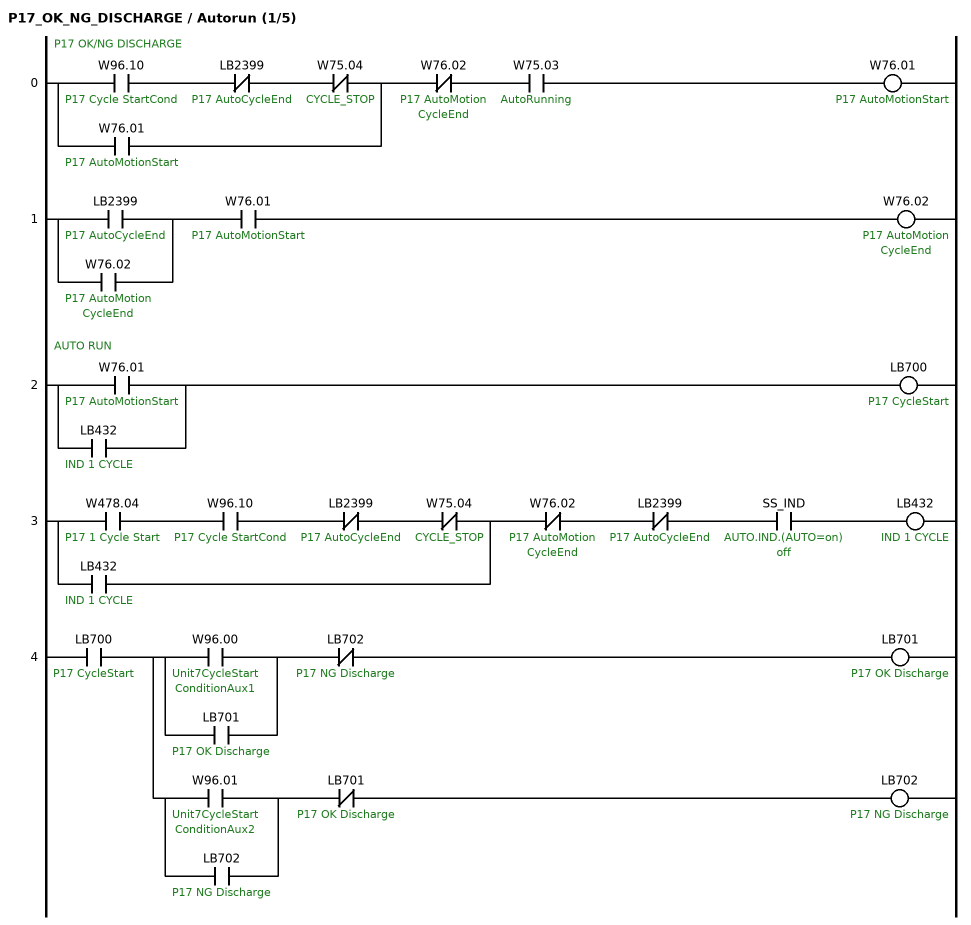
; rung 0: P17 OK/NG DISCHARGE
LD W96.10  ; P17 Cycle StartCond
ANDNOT LB2399  ; P17 AutoCycleEnd
ANDNOT W75.04  ; CYCLE_STOP
OR W76.01  ; P17 AutoMotionStart
ANDNOT W76.02  ; P17 AutoMotion CycleEnd
AND W75.03  ; AutoRunning
OUT W76.01  ; P17 AutoMotionStart
; rung 1
LD LB2399  ; P17 AutoCycleEnd
OR W76.02  ; P17 AutoMotion CycleEnd
AND W76.01  ; P17 AutoMotionStart
OUT W76.02  ; P17 AutoMotion CycleEnd
; rung 2: AUTO RUN
LD W76.01  ; P17 AutoMotionStart
OR LB432  ; IND 1 CYCLE
OUT LB700  ; P17 CycleStart
; rung 3
LD W478.04  ; P17 1 Cycle Start
AND W96.10  ; P17 Cycle StartCond
ANDNOT LB2399  ; P17 AutoCycleEnd
ANDNOT W75.04  ; CYCLE_STOP
OR LB432  ; IND 1 CYCLE
ANDNOT W76.02  ; P17 AutoMotion CycleEnd
ANDNOT LB2399  ; P17 AutoCycleEnd
AND SS_IND  ; AUTO.IND.(AUTO=on) off
OUT LB432  ; IND 1 CYCLE
; rung 4
LD LB700  ; P17 CycleStart
OUT TR0
LD W96.00  ; Unit7CycleStartConditionAux1
OR LB701  ; P17 OK Discharge
ANDLD
ANDNOT LB702  ; P17 NG Discharge
OUT LB701  ; P17 OK Discharge
LD TR0
LD W96.01  ; Unit7CycleStartConditionAux2
OR LB702  ; P17 NG Discharge
ANDLD
ANDNOT LB701  ; P17 OK Discharge
OUT LB702  ; P17 NG Discharge

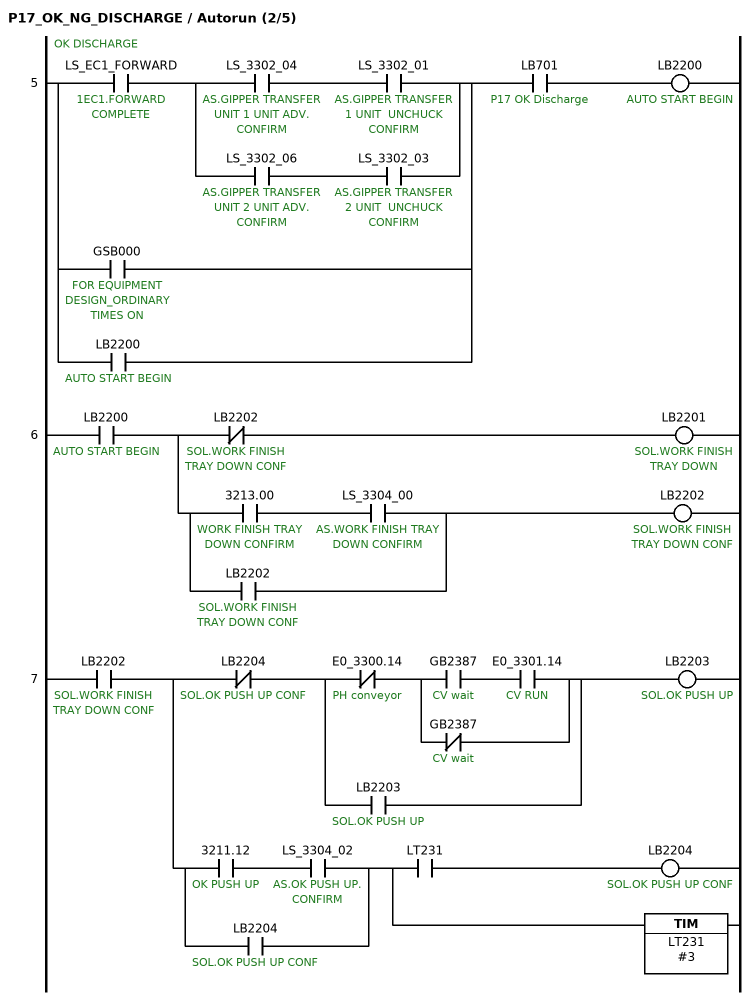
; rung 5: OK DISCHARGE
LD LS_EC1_FORWARD  ; 1EC1.FORWARD COMPLETE
LD LS_3302_04  ; AS.GIPPER TRANSFER UNIT 1 UNIT ADV. CONFIRM
AND LS_3302_01  ; AS.GIPPER TRANSFER 1 UNIT  UNCHUCK CONFIRM
LD LS_3302_06  ; AS.GIPPER TRANSFER UNIT 2 UNIT ADV. CONFIRM
AND LS_3302_03  ; AS.GIPPER TRANSFER 2 UNIT  UNCHUCK CONFIRM
ORLD
ANDLD
OR GSB000  ; FOR EQUIPMENT DESIGN_ORDINARY TIMES ON
OR LB2200  ; AUTO START BEGIN
AND LB701  ; P17 OK Discharge
OUT LB2200  ; AUTO START BEGIN
; rung 6
LD LB2200  ; AUTO START BEGIN
OUT TR0
ANDNOT LB2202  ; SOL.WORK FINISH TRAY DOWN CONF
OUT LB2201  ; SOL.WORK FINISH TRAY DOWN
LD TR0
LD 3213.00  ; WORK FINISH TRAY DOWN CONFIRM
AND LS_3304_00  ; AS.WORK FINISH TRAY DOWN CONFIRM
OR LB2202  ; SOL.WORK FINISH TRAY DOWN CONF
ANDLD
OUT LB2202  ; SOL.WORK FINISH TRAY DOWN CONF
; rung 7
LD LB2202  ; SOL.WORK FINISH TRAY DOWN CONF
OUT TR0
ANDNOT LB2204  ; SOL.OK PUSH UP CONF
LDNOT E0_3300.14  ; PH conveyor
LD GB2387  ; CV wait
AND E0_3301.14  ; CV RUN
ORNOT GB2387  ; CV wait
ANDLD
OR LB2203  ; SOL.OK PUSH UP
ANDLD
OUT LB2203  ; SOL.OK PUSH UP
LD TR0
LD 3211.12  ; OK PUSH UP
AND LS_3304_02  ; AS.OK PUSH UP. CONFIRM
OR LB2204  ; SOL.OK PUSH UP CONF
ANDLD
OUT TR0
AND LT231
OUT LB2204  ; SOL.OK PUSH UP CONF
LD TR0
TIM LT231 #3

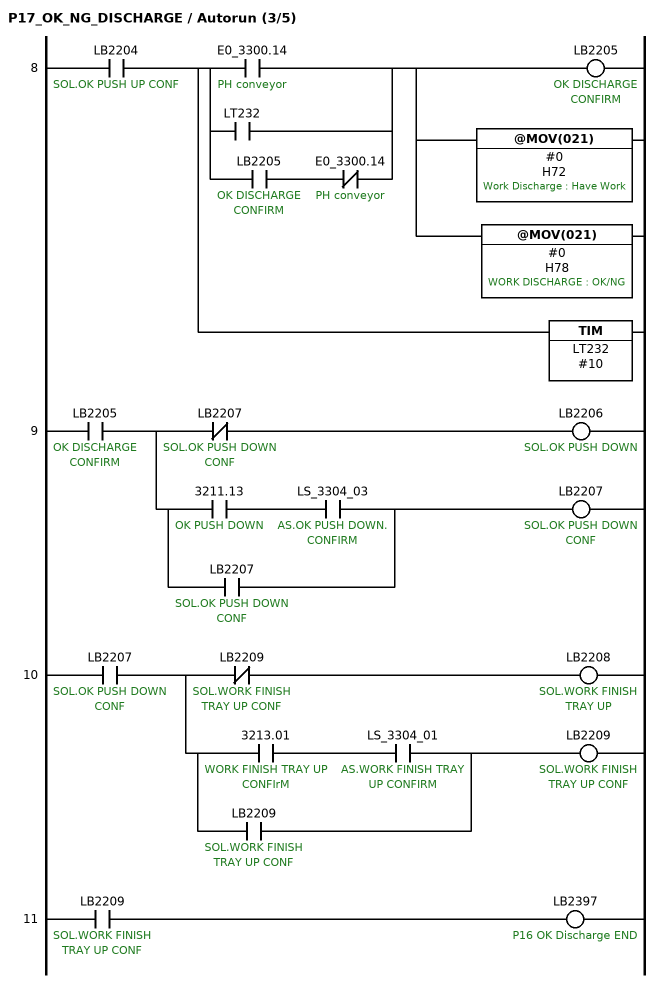
; rung 8
LD LB2204  ; SOL.OK PUSH UP CONF
OUT TR0
LD E0_3300.14  ; PH conveyor
OR LT232
LD LB2205  ; OK DISCHARGE CONFIRM
ANDNOT E0_3300.14  ; PH conveyor
ORLD
ANDLD
OUT LB2205  ; OK DISCHARGE CONFIRM
@MOV(021) #0 H72  ; Work Discharge : Have Work
@MOV(021) #0 H78  ; WORK DISCHARGE : OK/NG
LD TR0
TIM LT232 #10
; rung 9
LD LB2205  ; OK DISCHARGE CONFIRM
OUT TR0
ANDNOT LB2207  ; SOL.OK PUSH DOWN CONF
OUT LB2206  ; SOL.OK PUSH DOWN
LD TR0
LD 3211.13  ; OK PUSH DOWN
AND LS_3304_03  ; AS.OK PUSH DOWN. CONFIRM
OR LB2207  ; SOL.OK PUSH DOWN CONF
ANDLD
OUT LB2207  ; SOL.OK PUSH DOWN CONF
; rung 10
LD LB2207  ; SOL.OK PUSH DOWN CONF
OUT TR0
ANDNOT LB2209  ; SOL.WORK FINISH TRAY UP CONF
OUT LB2208  ; SOL.WORK FINISH TRAY UP
LD TR0
LD 3213.01  ; WORK FINISH TRAY UP CONFIrM
AND LS_3304_01  ; AS.WORK FINISH TRAY UP CONFIRM
OR LB2209  ; SOL.WORK FINISH TRAY UP CONF
ANDLD
OUT LB2209  ; SOL.WORK FINISH TRAY UP CONF
; rung 11
LD LB2209  ; SOL.WORK FINISH TRAY UP CONF
OUT LB2397  ; P16 OK Discharge END

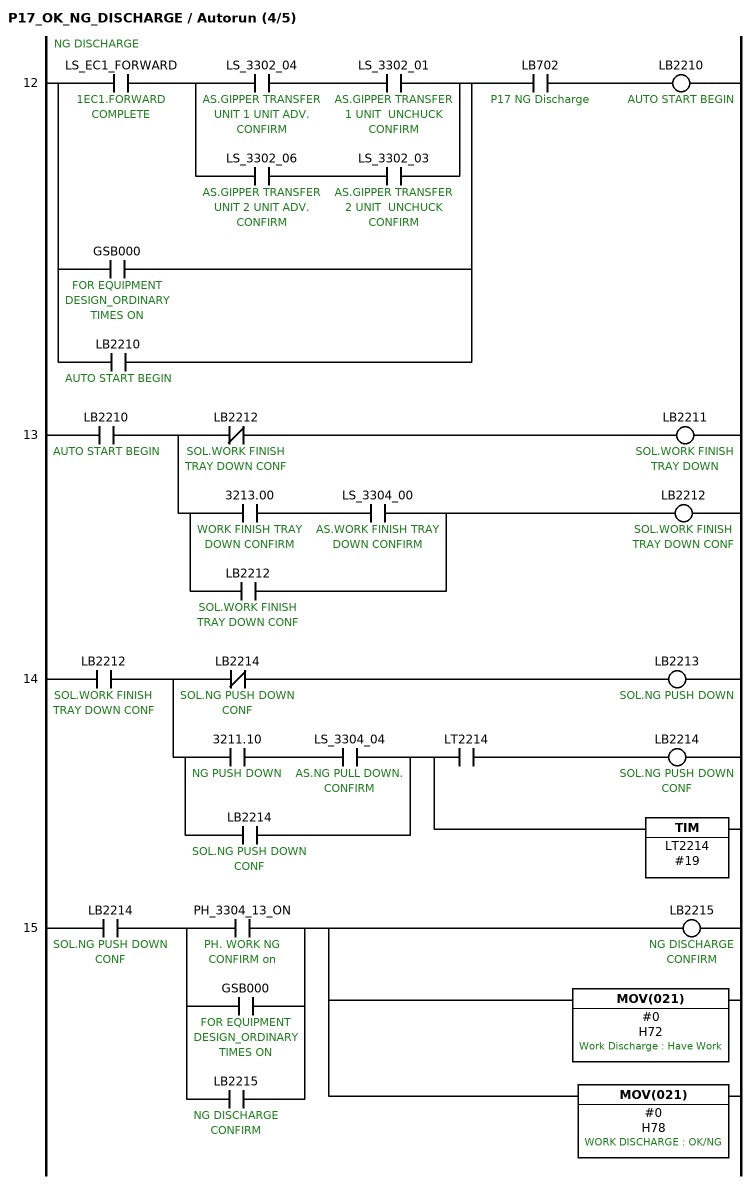
; rung 12: NG DISCHARGE
LD LS_EC1_FORWARD  ; 1EC1.FORWARD COMPLETE
LD LS_3302_04  ; AS.GIPPER TRANSFER UNIT 1 UNIT ADV. CONFIRM
AND LS_3302_01  ; AS.GIPPER TRANSFER 1 UNIT  UNCHUCK CONFIRM
LD LS_3302_06  ; AS.GIPPER TRANSFER UNIT 2 UNIT ADV. CONFIRM
AND LS_3302_03  ; AS.GIPPER TRANSFER 2 UNIT  UNCHUCK CONFIRM
ORLD
ANDLD
OR GSB000  ; FOR EQUIPMENT DESIGN_ORDINARY TIMES ON
OR LB2210  ; AUTO START BEGIN
AND LB702  ; P17 NG Discharge
OUT LB2210  ; AUTO START BEGIN
; rung 13
LD LB2210  ; AUTO START BEGIN
OUT TR0
ANDNOT LB2212  ; SOL.WORK FINISH TRAY DOWN CONF
OUT LB2211  ; SOL.WORK FINISH TRAY DOWN
LD TR0
LD 3213.00  ; WORK FINISH TRAY DOWN CONFIRM
AND LS_3304_00  ; AS.WORK FINISH TRAY DOWN CONFIRM
OR LB2212  ; SOL.WORK FINISH TRAY DOWN CONF
ANDLD
OUT LB2212  ; SOL.WORK FINISH TRAY DOWN CONF
; rung 14
LD LB2212  ; SOL.WORK FINISH TRAY DOWN CONF
OUT TR0
ANDNOT LB2214  ; SOL.NG PUSH DOWN CONF
OUT LB2213  ; SOL.NG PUSH DOWN
LD TR0
LD 3211.10  ; NG PUSH DOWN
AND LS_3304_04  ; AS.NG PULL DOWN. CONFIRM
OR LB2214  ; SOL.NG PUSH DOWN CONF
ANDLD
OUT TR0
AND LT2214
OUT LB2214  ; SOL.NG PUSH DOWN CONF
LD TR0
TIM LT2214 #19
; rung 15
LD LB2214  ; SOL.NG PUSH DOWN CONF
LD PH_3304_13_ON  ; PH. WORK NG CONFIRM on
OR GSB000  ; FOR EQUIPMENT DESIGN_ORDINARY TIMES ON
OR LB2215  ; NG DISCHARGE CONFIRM
ANDLD
OUT LB2215  ; NG DISCHARGE CONFIRM
MOV(021) #0 H72  ; Work Discharge : Have Work
MOV(021) #0 H78  ; WORK DISCHARGE : OK/NG

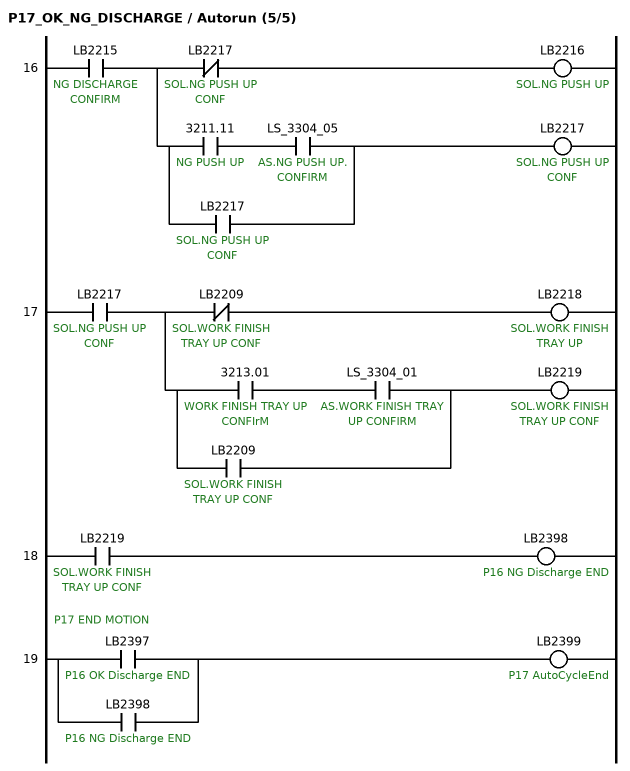
; rung 16
LD LB2215  ; NG DISCHARGE CONFIRM
OUT TR0
ANDNOT LB2217  ; SOL.NG PUSH UP CONF
OUT LB2216  ; SOL.NG PUSH UP
LD TR0
LD 3211.11  ; NG PUSH UP
AND LS_3304_05  ; AS.NG PUSH UP. CONFIRM
OR LB2217  ; SOL.NG PUSH UP CONF
ANDLD
OUT LB2217  ; SOL.NG PUSH UP CONF
; rung 17
LD LB2217  ; SOL.NG PUSH UP CONF
OUT TR0
ANDNOT LB2209  ; SOL.WORK FINISH TRAY UP CONF
OUT LB2218  ; SOL.WORK FINISH TRAY UP
LD TR0
LD 3213.01  ; WORK FINISH TRAY UP CONFIrM
AND LS_3304_01  ; AS.WORK FINISH TRAY UP CONFIRM
OR LB2209  ; SOL.WORK FINISH TRAY UP CONF
ANDLD
OUT LB2219  ; SOL.WORK FINISH TRAY UP CONF
; rung 18
LD LB2219  ; SOL.WORK FINISH TRAY UP CONF
OUT LB2398  ; P16 NG Discharge END
; rung 19: P17 END MOTION
LD LB2397  ; P16 OK Discharge END
OR LB2398  ; P16 NG Discharge END
OUT LB2399  ; P17 AutoCycleEnd

### Section Condition

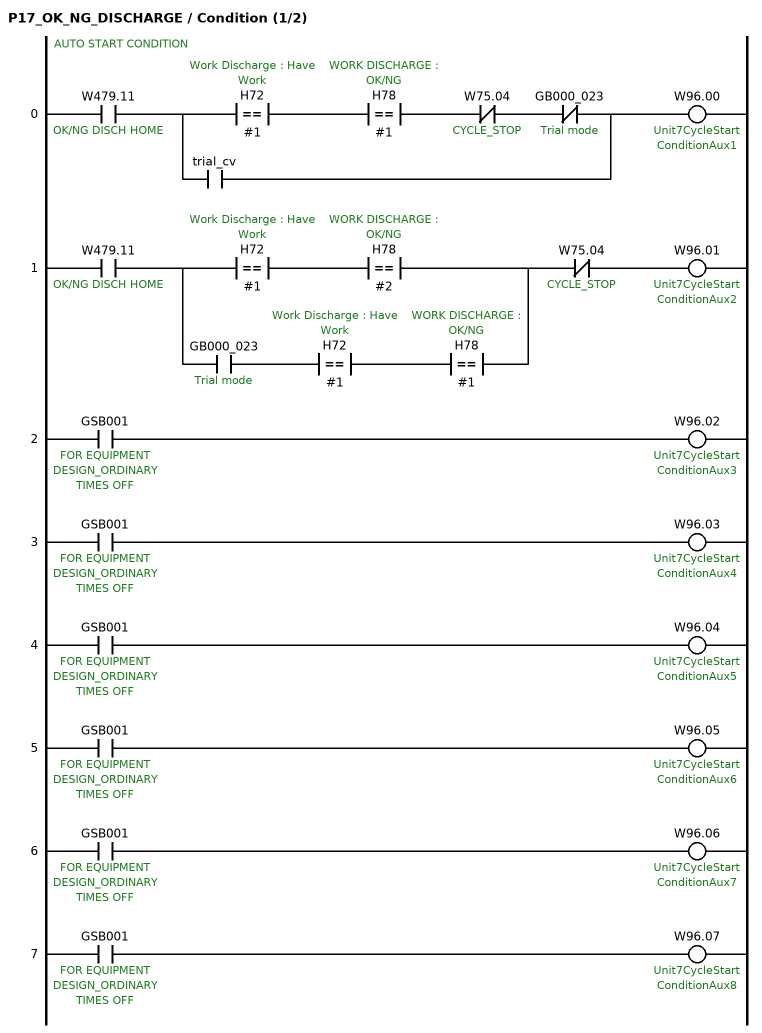
; rung 0: AUTO START CONDITION
LD W479.11  ; OK/NG DISCH HOME
LD=(300) H72 #1  ; Work Discharge : Have Work
AND=(300) H78 #1  ; WORK DISCHARGE : OK/NG
ANDNOT W75.04  ; CYCLE_STOP
ANDNOT GB000_023  ; Trial mode
OR trial_cv
ANDLD
OUT W96.00  ; Unit7CycleStartConditionAux1
; rung 1
LD W479.11  ; OK/NG DISCH HOME
LD=(300) H72 #1  ; Work Discharge : Have Work
AND=(300) H78 #2  ; WORK DISCHARGE : OK/NG
LD GB000_023  ; Trial mode
AND=(300) H72 #1  ; Work Discharge : Have Work
AND=(300) H78 #1  ; WORK DISCHARGE : OK/NG
ORLD
ANDLD
ANDNOT W75.04  ; CYCLE_STOP
OUT W96.01  ; Unit7CycleStartConditionAux2
; rung 2
LD GSB001  ; FOR EQUIPMENT DESIGN_ORDINARY TIMES OFF
OUT W96.02  ; Unit7CycleStartConditionAux3
; rung 3
LD GSB001  ; FOR EQUIPMENT DESIGN_ORDINARY TIMES OFF
OUT W96.03  ; Unit7CycleStartConditionAux4
; rung 4
LD GSB001  ; FOR EQUIPMENT DESIGN_ORDINARY TIMES OFF
OUT W96.04  ; Unit7CycleStartConditionAux5
; rung 5
LD GSB001  ; FOR EQUIPMENT DESIGN_ORDINARY TIMES OFF
OUT W96.05  ; Unit7CycleStartConditionAux6
; rung 6
LD GSB001  ; FOR EQUIPMENT DESIGN_ORDINARY TIMES OFF
OUT W96.06  ; Unit7CycleStartConditionAux7
; rung 7
LD GSB001  ; FOR EQUIPMENT DESIGN_ORDINARY TIMES OFF
OUT W96.07  ; Unit7CycleStartConditionAux8

